KUKA KRL program: MyProgram_073().src

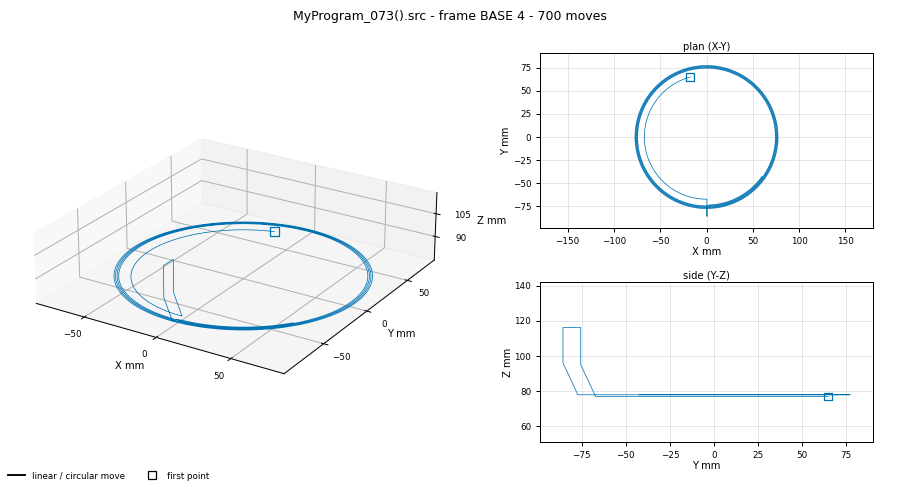
[picture p0: tool path of MyProgram_073().src in frame BASE 4, 700 of 700 moves have a stored position in this frame; points joined in program order, loops and branches not executed]
&ACCESS RVP
&REL 1
&PARAM TEMPLATE = C:\KRC\Roboter\Template\vorgabe
&PARAM EDITMASK = *
DEF MyProgram_073()
; ---- Setting reference (Base) ----
$BASE = BASE_DATA[4]

; --------------------------
; ---- Setting tool (TCP) ----
$TOOL = TOOL_DATA[3]
; --------------------------

$VEL.CP = VEL_APROX_PRINT
Startdeposition()
$VEL.CP = VEL_PRINT
LIN {X -17.4414,Y 64.8881,Z 77,A 99.3503,B 24.8705,C -2.6257,E1 24.9572,E2 344.7381} C_DIS
LIN {X -19.5195,Y 64.2946,Z 77,A 101.354,B 24.8704,C -2.6273,E1 24.9518,E2 342.7273} C_DIS
LIN {X -22.6182,Y 63.2711,Z 77,A 104.1504,B 24.8707,C -2.6243,E1 24.9445,E2 339.9329} C_DIS
LIN {X -25.654,Y 62.1019,Z 77,A 106.8913,B 24.8711,C -2.6198,E1 24.9374,E2 337.1966} C_DIS
LIN {X -27.9665,Y 61.0957,Z 77,A 109.0852,B 24.8714,C -2.6176,E1 24.9318,E2 335.0027} C_DIS
LIN {X -30.3307,Y 59.9565,Z 77,A 111.2597,B 24.8718,C -2.6126,E1 24.9263,E2 332.8342} C_DIS
LIN {X -32.9877,Y 58.5366,Z 77,A 113.6029,B 24.8728,C -2.6034,E1 24.9206,E2 330.5064} C_DIS
LIN {X -35.1348,Y 57.2737,Z 77,A 115.7355,B 24.8731,C -2.5997,E1 24.9155,E2 328.3759} C_DIS
LIN {X -37.2111,Y 55.947,Z 77,A 117.8448,B 24.8735,C -2.596,E1 24.9106,E2 326.2688} C_DIS
LIN {X -38.795,Y 54.8606,Z 77,A 119.7284,B 24.8733,C -2.598,E1 24.9063,E2 324.3738} C_DIS
LIN {X -41.2648,Y 53.028,Z 77,A 122.3339,B 24.8738,C -2.5922,E1 24.9005,E2 321.7728} C_DIS
LIN {X -43.4924,Y 51.216,Z 77,A 124.7333,B 24.8745,C -2.5859,E1 24.8953,E2 319.3795} C_DIS
LIN {X -45.7228,Y 49.2366,Z 77,A 127.4573,B 24.8747,C -2.5839,E1 24.8897,E2 316.6491} C_DIS
LIN {X -48.0153,Y 47.0029,Z 77,A 130.0891,B 24.8755,C -2.5754,E1 24.8845,E2 314.0265} C_DIS
LIN {X -50.0114,Y 44.8723,Z 77,A 132.6532,B 24.8759,C -2.5708,E1 24.8797,E2 311.462} C_DIS
LIN {X -51.9391,Y 42.6281,Z 77,A 135.2435,B 24.8764,C -2.5658,E1 24.875,E2 308.8718} C_DIS
LIN {X -53.955,Y 40.0458,Z 77,A 138.0531,B 24.8771,C -2.5588,E1 24.8703,E2 306.0656} C_DIS
LIN {X -55.8378,Y 37.3755,Z 77,A 140.854,B 24.8778,C -2.5515,E1 24.8659,E2 303.2682} C_DIS
LIN {X -57.2778,Y 35.128,Z 77,A 143.0663,B 24.8785,C -2.5438,E1 24.8626,E2 301.063} C_DIS
LIN {X -58.5282,Y 33.0027,Z 77,A 145.1855,B 24.8791,C -2.5382,E1 24.8597,E2 298.9463} C_DIS
LIN {X -59.947,Y 30.3494,Z 77,A 147.5323,B 24.8802,C -2.5262,E1 24.8566,E2 296.6154} C_DIS
LIN {X -61.0193,Y 28.1312,Z 77,A 149.6529,B 24.8808,C -2.5204,E1 24.8541,E2 294.4971} C_DIS
LIN {X -61.8116,Y 26.3449,Z 77,A 151.5592,B 24.8808,C -2.5204,E1 24.852,E2 292.5804} C_DIS
LIN {X -62.8919,Y 23.6492,Z 77,A 153.9533,B 24.8816,C -2.5112,E1 24.8496,E2 290.1948} C_DIS
LIN {X -63.8037,Y 21.0691,Z 77,A 156.4499,B 24.882,C -2.5074,E1 24.8473,E2 287.6931} C_DIS
LIN {X -64.5709,Y 18.583,Z 77,A 158.637,B 24.8827,C -2.4999,E1 24.8456,E2 285.5113} C_DIS
LIN {X -65.3372,Y 15.6772,Z 77,A 161.2488,B 24.8833,C -2.4929,E1 24.8438,E2 282.9009} C_DIS
LIN {X -65.9008,Y 13.1111,Z 77,A 163.5551,B 24.8839,C -2.4872,E1 24.8425,E2 280.5947} C_DIS
LIN {X -66.4404,Y 10.0194,Z 77,A 166.0408,B 24.885,C -2.4749,E1 24.8414,E2 278.1237} C_DIS
LIN {X -66.7829,Y 7.4076,Z 77,A 168.5127,B 24.8853,C -2.4724,E1 24.8406,E2 275.6429} C_DIS
LIN {X -67.0644,Y 4.1441,Z 77,A 171.3257,B 24.8861,C -2.4639,E1 24.84,E2 272.8332} C_DIS
LIN {X -67.1864,Y 0.8793,Z 77,A 174.1109,B 24.8869,C -2.4551,E1 24.8398,E2 270.0523} C_DIS
LIN {X -67.1706,Y -1.7002,Z 77,A 176.322,B 24.8875,C -2.4484,E1 24.8398,E2 267.844} C_DIS
LIN {X -67.01,Y -4.9472,Z 77,A 178.9028,B 24.8887,C -2.4357,E1 24.8403,E2 265.2779} C_DIS
LIN {X -66.7829,Y -7.4069,Z 77,A -178.7682,B 24.8888,C -2.4337,E1 24.841,E2 262.9398} C_DIS
LIN {X -66.4656,Y -9.8566,Z 77,A -176.8004,B 24.8897,C -2.4243,E1 24.8417,E2 260.9827} C_DIS
LIN {X -66.0524,Y -12.3243,Z 77,A -174.473,B 24.8899,C -2.4218,E1 24.8429,E2 258.6476} C_DIS
LIN {X -65.4042,Y -15.3955,Z 77,A -171.9941,B 24.891,C -2.4095,E1 24.8444,E2 256.1833} C_DIS
LIN {X -64.7607,Y -17.9129,Z 77,A -169.5742,B 24.8913,C -2.4071,E1 24.8461,E2 253.7552} C_DIS
LIN {X -64.0539,Y -20.2957,Z 77,A -167.6468,B 24.8922,C -2.3968,E1 24.8477,E2 251.8412} C_DIS
LIN {X -63.2656,Y -22.6337,Z 77,A -165.321,B 24.8923,C -2.3953,E1 24.8498,E2 249.5058} C_DIS
LIN {X -62.3396,Y -25.07,Z 77,A -163.1316,B 24.893,C -2.3883,E1 24.8521,E2 247.321} C_DIS
LIN {X -61.1455,Y -27.8561,Z 77,A -160.6723,B 24.8939,C -2.3784,E1 24.8548,E2 244.8718} C_DIS
LIN {X -60.0186,Y -30.2091,Z 77,A -158.2271,B 24.8939,C -2.3769,E1 24.8579,E2 242.417} C_DIS
LIN {X -58.6544,Y -32.7767,Z 77,A -155.7358,B 24.8946,C -2.3705,E1 24.8612,E2 239.9277} C_DIS
LIN {X -57.2052,Y -35.2475,Z 77,A -153.2924,B 24.8951,C -2.3642,E1 24.8647,E2 237.4869} C_DIS
LIN {X -55.7951,Y -37.4385,Z 77,A -151.1058,B 24.8957,C -2.3578,E1 24.8681,E2 235.3045} C_DIS
LIN {X -54.384,Y -39.4603,Z 77,A -148.9837,B 24.8961,C -2.3531,E1 24.8715,E2 233.1833} C_DIS
LIN {X -52.5036,Y -41.9302,Z 77,A -146.3519,B 24.8967,C -2.3465,E1 24.876,E2 230.5548} C_DIS
LIN {X -51.184,Y -43.53,Z 77,A -144.6169,B 24.8971,C -2.3418,E1 24.8791,E2 228.8231} C_DIS
LIN {X -49.2273,Y -45.7329,Z 77,A -141.9644,B 24.8973,C -2.3393,E1 24.8841,E2 226.1648} C_DIS
LIN {X -47.2236,Y -47.7973,Z 77,A -139.6629,B 24.8981,C -2.3309,E1 24.8886,E2 223.8736} C_DIS
LIN {X -45.1372,Y -49.774,Z 77,A -137.1132,B 24.8983,C -2.3281,E1 24.8939,E2 221.32} C_DIS
LIN {X -42.9447,Y -51.676,Z 77,A -134.7116,B 24.8988,C -2.3219,E1 24.899,E2 218.9241} C_DIS
LIN {X -40.6905,Y -53.4706,Z 77,A -132.0959,B 24.8989,C -2.321,E1 24.9047,E2 216.3008} C_DIS
LIN {X -38.6866,Y -54.9378,Z 77,A -129.9758,B 24.8992,C -2.3175,E1 24.9096,E2 214.1817} C_DIS
LIN {X -36.6463,Y -56.3194,Z 77,A -127.8662,B 24.8995,C -2.3145,E1 24.9145,E2 212.0724} C_DIS
LIN {X -34.5571,Y -57.6248,Z 77,A -125.8772,B 24.9,C -2.3089,E1 24.9192,E2 210.0906} C_DIS
LIN {X -32.3987,Y -58.8655,Z 77,A -123.6283,B 24.9,C -2.3089,E1 24.9247,E2 207.8352} C_DIS
LIN {X -30.2145,Y -60.0159,Z 77,A -121.5171,B 24.9002,C -2.3064,E1 24.9299,E2 205.7242} C_DIS
LIN {X -27.8627,Y -61.1425,Z 77,A -119.3351,B 24.9005,C -2.3029,E1 24.9355,E2 203.5449} C_DIS
LIN {X -25.0759,Y -62.3372,Z 77,A -116.8865,B 24.901,C -2.2972,E1 24.9418,E2 201.1044} C_DIS
LIN {X -22.6444,Y -63.2618,Z 77,A -114.4748,B 24.9008,C -2.2997,E1 24.9481,E2 198.6819} C_DIS
LIN {X -20.312,Y -64.0487,Z 77,A -112.5912,B 24.9013,C -2.2931,E1 24.9531,E2 196.8105} C_DIS
LIN {X -17.9227,Y -64.758,Z 77,A -110.242,B 24.901,C -2.2969,E1 24.9594,E2 194.4485} C_DIS
LIN {X -15.3953,Y -65.4043,Z 77,A -108.0635,B 24.9012,C -2.2947,E1 24.9653,E2 192.2723} C_DIS
LIN {X -12.4424,Y -66.0296,Z 77,A -105.7199,B 24.9018,C -2.2882,E1 24.9717,E2 189.9414} C_DIS
LIN {X -9.9977,Y -66.4438,Z 77,A -103.6077,B 24.9018,C -2.2876,E1 24.9775,E2 187.8287} C_DIS
LIN {X -7.5502,Y -66.7662,Z 77,A -101.2755,B 24.9014,C -2.2926,E1 24.984,E2 185.4829} C_DIS
LIN {X -4.954,Y -67.0095,Z 77,A -99.2056,B 24.9017,C -2.2889,E1 24.9898,E2 183.421} C_DIS
LIN {X -2.4711,Y -67.147,Z 77,A -96.8737,B 24.9013,C -2.2941,E1 24.9963,E2 181.076} C_DIS
LIN {X 0.4221,Y -67.1891,Z 77,A -94.9568,B 24.9024,C -2.2814,E1 25.0016,E2 179.1893} C_DIS
Enddeposition()
LIN {X 0.4386,Y -69.3021,Z 81.5315,A -94.9475,B 24.9027,C -2.2775,E1 25.0016,E2 179.1893} C_DIS
LIN {X 0.4882,Y -75.6412,Z 95.1262,A -94.9245,B 24.9035,C -2.2678,E1 25.0016,E2 179.1893} C_DIS
LIN {X 0.4882,Y -75.6412,Z 116.1262,A -95.2835,B 24.8902,C -2.4189,E1 25.0016,E2 179.1893} C_DIS
LIN {X 0.5081,Y -85.7186,Z 116.1262,A -95.3115,B 24.9057,C -2.2421,E1 25.0003,E2 179.6373} C_DIS
LIN {X 0.5081,Y -85.7186,Z 96.1262,A -94.9701,B 24.9174,C -2.0983,E1 25.0003,E2 179.6373} C_DIS
LIN {X 0.5081,Y -79.3793,Z 82.5315,A -94.9916,B 24.9167,C -2.1074,E1 25.0003,E2 179.6373} C_DIS
LIN {X 0.5081,Y -77.2663,Z 78,A -95.0003,B 24.9164,C -2.111,E1 25.0003,E2 179.6373} C_DIS
Startdeposition()
$VEL.CP = VEL_PRINT
LIN {X 3.5724,Y -77.1871,Z 78,A -91.8935,B 24.9145,C -2.1352,E1 25.0091,E2 176.4739} C_DIS
LIN {X 6.411,Y -77.0033,Z 78,A -89.9101,B 24.9147,C -2.1326,E1 25.0146,E2 174.4976} C_DIS
LIN {X 8.7348,Y -76.7744,Z 78,A -88.2092,B 24.9147,C -2.1326,E1 25.0194,E2 172.7976} C_DIS
LIN {X 10.6163,Y -76.5369,Z 78,A -86.6281,B 24.9142,C -2.1386,E1 25.0238,E2 171.2038} C_DIS
LIN {X 13.2103,Y -76.1331,Z 78,A -84.738,B 24.9142,C -2.1384,E1 25.029,E2 169.316} C_DIS
LIN {X 15.7888,Y -75.6394,Z 78,A -82.8059,B 24.9142,C -2.1396,E1 25.0343,E2 167.3833} C_DIS
LIN {X 18.0671,Y -75.1278,Z 78,A -80.9865,B 24.9138,C -2.1438,E1 25.0392,E2 165.5566} C_DIS
LIN {X 20.8201,Y -74.4119,Z 78,A -78.9095,B 24.9137,C -2.1451,E1 25.0448,E2 163.4798} C_DIS
LIN {X 23.3362,Y -73.6626,Z 78,A -77.0207,B 24.9137,C -2.1457,E1 25.0499,E2 161.5932} C_DIS
LIN {X 25.9989,Y -72.7653,Z 78,A -75.0657,B 24.9137,C -2.1445,E1 25.055,E2 159.6447} C_DIS
LIN {X 27.8093,Y -72.093,Z 78,A -73.5154,B 24.9133,C -2.1499,E1 25.0591,E2 158.085} C_DIS
LIN {X 29.7724,Y -71.3037,Z 78,A -72.0267,B 24.9133,C -2.1499,E1 25.0629,E2 156.6} C_DIS
LIN {X 32.1778,Y -70.2521,Z 78,A -69.914,B 24.9127,C -2.1576,E1 25.0683,E2 154.4739} C_DIS
LIN {X 34.7418,Y -69.0201,Z 78,A -67.9092,B 24.9127,C -2.1579,E1 25.0733,E2 152.4738} C_DIS
LIN {X 37.0659,Y -67.7992,Z 78,A -66.0648,B 24.9127,C -2.1582,E1 25.0779,E2 150.6339} C_DIS
LIN {X 38.9088,Y -66.7598,Z 78,A -64.5303,B 24.9125,C -2.16,E1 25.0816,E2 149.0999} C_DIS
LIN {X 40.7215,Y -65.6686,Z 78,A -62.792,B 24.9118,C -2.168,E1 25.0858,E2 147.3481} C_DIS
LIN {X 43.1109,Y -64.1253,Z 78,A -60.6916,B 24.9115,C -2.1718,E1 25.0907,E2 145.2456} C_DIS
LIN {X 45.265,Y -62.6246,Z 78,A -58.8065,B 24.9114,C -2.1739,E1 25.095,E2 143.3622} C_DIS
LIN {X 47.3656,Y -61.05,Z 78,A -56.7925,B 24.9109,C -2.1801,E1 25.0994,E2 141.3409} C_DIS
LIN {X 49.7493,Y -59.125,Z 78,A -54.6079,B 24.9107,C -2.1824,E1 25.1041,E2 139.1592} C_DIS
LIN {X 51.7284,Y -57.4001,Z 78,A -52.6061,B 24.9102,C -2.1885,E1 25.1083,E2 137.1508} C_DIS
LIN {X 53.964,Y -55.305,Z 78,A -50.411,B 24.9099,C -2.1915,E1 25.1128,E2 134.9576} C_DIS
LIN {X 55.4573,Y -53.8061,Z 78,A -48.9275,B 24.9099,C -2.1928,E1 25.1157,E2 133.4776} C_DIS
LIN {X 57.2538,Y -51.8918,Z 78,A -47.0377,B 24.9096,C -2.1959,E1 25.1192,E2 131.5887} C_DIS
LIN {X 58.5101,Y -50.4711,Z 78,A -45.6394,B 24.9093,C -2.1992,E1 25.1218,E2 130.1889} C_DIS
LIN {X 59.8692,Y -48.8496,Z 78,A -44.0797,B 24.909,C -2.203,E1 25.1246,E2 128.6273} C_DIS
LIN {X 61.05,Y -47.3656,Z 78,A -42.5054,B 24.9082,C -2.2119,E1 25.1273,E2 127.0395} C_DIS
LIN {X 62.6246,Y -45.265,Z 78,A -40.495,B 24.9076,C -2.2191,E1 25.1307,E2 125.0218} C_DIS
LIN {X 64.369,Y -42.7462,Z 78,A -38.4884,B 24.9078,C -2.2172,E1 25.1338,E2 123.0295} C_DIS
LIN {X 65.6686,Y -40.7215,Z 78,A -36.5637,B 24.907,C -2.2266,E1 25.1367,E2 121.0924} C_DIS
LIN {X 66.8691,Y -38.7186,Z 78,A -34.9946,B 24.907,C -2.2265,E1 25.1389,E2 119.5316} C_DIS
LIN {X 67.7992,Y -37.0659,Z 78,A -33.4212,B 24.9062,C -2.2357,E1 25.141,E2 117.9446} C_DIS
LIN {X 69.1843,Y -34.4106,Z 78,A -31.2395,B 24.9058,C -2.241,E1 25.1438,E2 115.7619} C_DIS
LIN {X 70.2521,Y -32.1778,Z 78,A -29.5677,B 24.9058,C -2.2414,E1 25.1458,E2 114.0982} C_DIS
LIN {X 71.0206,Y -30.4441,Z 78,A -28.1708,B 24.9054,C -2.2454,E1 25.1473,E2 112.6997} C_DIS
LIN {X 71.8265,Y -28.4878,Z 78,A -26.6126,B 24.905,C -2.2498,E1 25.149,E2 111.1396} C_DIS
LIN {X 72.6786,Y -26.2378,Z 78,A -24.8119,B 24.9045,C -2.2558,E1 25.1507,E2 109.3348} C_DIS
LIN {X 73.4383,Y -24.0297,Z 78,A -23.1208,B 24.9042,C -2.2599,E1 25.1522,E2 107.6437} C_DIS
LIN {X 74.0325,Y -22.1305,Z 78,A -21.4792,B 24.9034,C -2.2696,E1 25.1536,E2 105.9883} C_DIS
LIN {X 74.7736,Y -19.4812,Z 78,A -19.4536,B 24.9029,C -2.2756,E1 25.155,E2 103.9604} C_DIS
LIN {X 75.3932,Y -16.9301,Z 78,A -17.5731,B 24.9025,C -2.2796,E1 25.1562,E2 102.0812} C_DIS
LIN {X 75.9238,Y -14.359,Z 78,A -15.7346,B 24.9023,C -2.2824,E1 25.1572,E2 100.2468} C_DIS
LIN {X 76.323,Y -12.0583,Z 78,A -13.8679,B 24.9014,C -2.2921,E1 25.1581,E2 98.3681} C_DIS
LIN {X 76.6896,Y -9.4588,Z 78,A -11.9876,B 24.9011,C -2.2962,E1 25.1587,E2 96.4893} C_DIS
LIN {X 76.9188,Y -7.3554,Z 78,A -10.3392,B 24.9004,C -2.3037,E1 25.1592,E2 94.8329} C_DIS
LIN {X 77.1468,Y -4.3496,Z 78,A -8.1686,B 24.9,C -2.3089,E1 25.1596,E2 92.6631} C_DIS
LIN {X 77.2649,Y -0.9482,Z 78,A -5.7244,B 24.8995,C -2.3144,E1 25.1598,E2 90.2204} C_DIS
LIN {X 77.2557,Y 1.4489,Z 78,A -3.9631,B 24.8991,C -2.3196,E1 25.1598,E2 88.4573} C_DIS
LIN {X 77.1655,Y 4.0105,Z 78,A -2.1749,B 24.8988,C -2.3221,E1 25.1595,E2 86.6738} C_DIS
LIN {X 77.0033,Y 6.411,Z 78,A -0.3747,B 24.8983,C -2.3282,E1 25.1591,E2 84.8698} C_DIS
LIN {X 76.7744,Y 8.7348,Z 78,A 1.3165,B 24.8979,C -2.3324,E1 25.1586,E2 83.1787} C_DIS
LIN {X 76.5369,Y 10.6163,Z 78,A 2.7127,B 24.8976,C -2.3365,E1 25.1581,E2 81.7811} C_DIS
LIN {X 76.1693,Y 12.994,Z 78,A 4.6361,B 24.8967,C -2.3464,E1 25.1573,E2 79.8457} C_DIS
LIN {X 75.6394,Y 15.7888,Z 78,A 6.6081,B 24.8965,C -2.3486,E1 25.1562,E2 77.8799} C_DIS
LIN {X 75.0434,Y 18.413,Z 78,A 8.7541,B 24.8955,C -2.3593,E1 25.1548,E2 75.7209} C_DIS
LIN {X 74.4119,Y 20.8201,Z 78,A 10.5707,B 24.8951,C -2.364,E1 25.1535,E2 73.9038} C_DIS
LIN {X 73.6626,Y 23.3362,Z 78,A 12.4518,B 24.8948,C -2.3678,E1 25.1519,E2 72.0245} C_DIS
LIN {X 72.8689,Y 25.7037,Z 78,A 14.3528,B 24.8942,C -2.3748,E1 25.1502,E2 70.1177} C_DIS
LIN {X 71.8089,Y 28.5327,Z 78,A 16.536,B 24.8938,C -2.3795,E1 25.148,E2 67.9355} C_DIS
LIN {X 70.9329,Y 30.6451,Z 78,A 18.1646,B 24.8935,C -2.3822,E1 25.1462,E2 66.3093} C_DIS
LIN {X 69.8519,Y 33.0375,Z 78,A 20.0137,B 24.8933,C -2.3847,E1 25.1441,E2 64.4644} C_DIS
LIN {X 69.0201,Y 34.7418,Z 78,A 21.5348,B 24.8926,C -2.3921,E1 25.1422,E2 62.9339} C_DIS
LIN {X 67.7992,Y 37.0659,Z 78,A 23.4982,B 24.8921,C -2.3979,E1 25.1396,E2 60.9672} C_DIS
LIN {X 66.3889,Y 39.5363,Z 78,A 25.5956,B 24.8916,C -2.4031,E1 25.1366,E2 58.8683} C_DIS
LIN {X 65.164,Y 41.5242,Z 78,A 27.3414,B 24.8912,C -2.408,E1 25.134,E2 57.1197} C_DIS
LIN {X 63.5914,Y 43.8946,Z 78,A 29.2628,B 24.8912,C -2.4076,E1 25.131,E2 55.2087} C_DIS
LIN {X 62.1567,Y 45.904,Z 78,A 31.099,B 24.8908,C -2.4123,E1 25.128,E2 53.3704} C_DIS
LIN {X 60.9161,Y 47.5394,Z 78,A 32.5976,B 24.8905,C -2.4152,E1 25.1255,E2 51.8719} C_DIS
LIN {X 59.5909,Y 49.1887,Z 78,A 34.1584,B 24.8902,C -2.4186,E1 25.1227,E2 50.3103} C_DIS
LIN {X 58.0306,Y 51.0201,Z 78,A 36.0854,B 24.8895,C -2.427,E1 25.1192,E2 48.3723} C_DIS
LIN {X 56.1134,Y 53.1215,Z 78,A 38.1845,B 24.8891,C -2.4313,E1 25.1152,E2 46.2722} C_DIS
LIN {X 54.0086,Y 55.261,Z 78,A 40.2505,B 24.8891,C -2.4313,E1 25.1111,E2 44.2151} C_DIS
LIN {X 52.5905,Y 56.6127,Z 78,A 41.6938,B 24.8888,C -2.4339,E1 25.1082,E2 42.7713} C_DIS
LIN {X 51.1853,Y 57.8863,Z 78,A 43.094,B 24.8886,C -2.4365,E1 25.1053,E2 41.3707} C_DIS
LIN {X 49.5806,Y 59.2652,Z 78,A 44.8414,B 24.8878,C -2.4447,E1 25.1015,E2 39.6104} C_DIS
LIN {X 47.5394,Y 60.9161,Z 78,A 46.5952,B 24.888,C -2.4426,E1 25.0977,E2 37.8683} C_DIS
LIN {X 46.0301,Y 62.0644,Z 78,A 48.1194,B 24.8875,C -2.4485,E1 25.0943,E2 36.3356} C_DIS
LIN {X 44.313,Y 63.3006,Z 78,A 49.7356,B 24.8871,C -2.4525,E1 25.0906,E2 34.7154} C_DIS
LIN {X 41.9531,Y 64.8887,Z 78,A 51.8709,B 24.8867,C -2.4566,E1 25.0856,E2 32.5775} C_DIS
LIN {X 39.5363,Y 66.3889,Z 78,A 53.9546,B 24.8865,C -2.459,E1 25.0806,E2 30.4946} C_DIS
LIN {X 37.0659,Y 67.7992,Z 78,A 56.0713,B 24.8862,C -2.4621,E1 25.0755,E2 28.3768} C_DIS
LIN {X 34.7418,Y 69.0201,Z 78,A 57.9311,B 24.8862,C -2.4621,E1 25.0708,E2 26.5222} C_DIS
LIN {X 32.3767,Y 70.1595,Z 78,A 59.7773,B 24.8862,C -2.4615,E1 25.0662,E2 24.6822} C_DIS
LIN {X 30.214,Y 71.1176,Z 78,A 61.7043,B 24.8856,C -2.4684,E1 25.0612,E2 22.7435} C_DIS
LIN {X 27.6042,Y 72.1707,Z 78,A 63.7884,B 24.8855,C -2.4703,E1 25.0558,E2 20.6594} C_DIS
LIN {X 25.137,Y 73.0678,Z 78,A 65.6828,B 24.8855,C -2.4705,E1 25.0508,E2 18.7684} C_DIS
LIN {X 22.4305,Y 73.9435,Z 78,A 67.6298,B 24.8857,C -2.4675,E1 25.0457,E2 16.832} C_DIS
LIN {X 20.4809,Y 74.5063,Z 78,A 69.1796,B 24.8855,C -2.4698,E1 25.0415,E2 15.2793} C_DIS
LIN {X 18.0671,Y 75.1278,Z 78,A 71.1302,B 24.8851,C -2.4738,E1 25.0362,E2 13.3222} C_DIS
LIN {X 15.7888,Y 75.6394,Z 78,A 72.8846,B 24.8851,C -2.4752,E1 25.0314,E2 11.5666} C_DIS
LIN {X 13.2103,Y 76.1331,Z 78,A 74.8861,B 24.8848,C -2.4775,E1 25.0259,E2 9.562} C_DIS
LIN {X 10.3991,Y 76.5678,Z 78,A 76.7607,B 24.8854,C -2.4715,E1 25.0208,E2 7.7033} C_DIS
LIN {X 8.2988,Y 76.8227,Z 78,A 78.4702,B 24.885,C -2.4757,E1 25.016,E2 5.9851} C_DIS
LIN {X 5.6844,Y 77.0614,Z 78,A 80.2757,B 24.8853,C -2.4719,E1 25.011,E2 4.1896} C_DIS
LIN {X 3.5724,Y 77.1871,Z 78,A 82.0378,B 24.8848,C -2.4772,E1 25.006,E2 2.4156} C_DIS
LIN {X 0.7289,Y 77.2663,Z 78,A 84.134,B 24.8848,C -2.4765,E1 25.0002,E2 0.3211} C_DIS
LIN {X -2.1156,Y 77.2407,Z 78,A 86.2424,B 24.8849,C -2.476,E1 24.9943,E2 -1.7861} C_DIS
LIN {X -4.9571,Y 77.1105,Z 78,A 88.3533,B 24.885,C -2.4752,E1 24.9884,E2 -3.8959} C_DIS
LIN {X -7.5739,Y 76.8986,Z 78,A 90.3728,B 24.885,C -2.4763,E1 24.9828,E2 -5.9188} C_DIS
LIN {X -10.6163,Y 76.5369,Z 78,A 92.5774,B 24.8852,C -2.4731,E1 24.9767,E2 -8.1174} C_DIS
LIN {X -13.2103,Y 76.1331,Z 78,A 94.5292,B 24.8853,C -2.4718,E1 24.9713,E2 -10.0681} C_DIS
LIN {X -16.0036,Y 75.5953,Z 78,A 96.4626,B 24.8859,C -2.4654,E1 24.9661,E2 -11.9884} C_DIS
LIN {X -18.0671,Y 75.1278,Z 78,A 98.2126,B 24.8856,C -2.4688,E1 24.9613,E2 -13.7489} C_DIS
LIN {X -20.8201,Y 74.4119,Z 78,A 100.3265,B 24.8858,C -2.4668,E1 24.9556,E2 -15.8612} C_DIS
LIN {X -23.3465,Y 73.6593,Z 78,A 102.2266,B 24.8861,C -2.4631,E1 24.9506,E2 -17.7559} C_DIS
LIN {X -25.3439,Y 72.9951,Z 78,A 103.6735,B 24.8866,C -2.4583,E1 24.9467,E2 -19.194} C_DIS
LIN {X -27.6042,Y 72.1707,Z 78,A 105.6159,B 24.8864,C -2.4601,E1 24.9416,E2 -21.1448} C_DIS
LIN {X -29.7724,Y 71.3037,Z 78,A 107.3776,B 24.8866,C -2.4585,E1 24.9371,E2 -22.9066} C_DIS
LIN {X -32.3767,Y 70.1595,Z 78,A 109.4937,B 24.8868,C -2.4556,E1 24.9317,E2 -25.0208} C_DIS
LIN {X -34.7418,Y 69.0201,Z 78,A 111.5353,B 24.8868,C -2.4549,E1 24.9266,E2 -27.0663} C_DIS
LIN {X -37.4502,Y 67.5876,Z 78,A 113.7281,B 24.8874,C -2.4491,E1 24.9212,E2 -29.2513} C_DIS
LIN {X -39.7251,Y 66.2773,Z 78,A 115.6291,B 24.8879,C -2.4444,E1 24.9167,E2 -31.1469} C_DIS
LIN {X -41.9531,Y 64.8887,Z 78,A 117.6129,B 24.8881,C -2.4418,E1 24.912,E2 -33.1307} C_DIS
LIN {X -44.313,Y 63.3006,Z 78,A 119.6067,B 24.8888,C -2.4347,E1 24.9074,E2 -35.1145} C_DIS
LIN {X -46.2055,Y 61.9327,Z 78,A 121.4956,B 24.8888,C -2.4352,E1 24.9032,E2 -37.0111} C_DIS
LIN {X -48.4538,Y 60.19,Z 78,A 123.4366,B 24.8895,C -2.4264,E1 24.8989,E2 -38.9385} C_DIS
LIN {X -49.9163,Y 58.9828,Z 78,A 125.017,B 24.8894,C -2.4277,E1 24.8955,E2 -40.5281} C_DIS
LIN {X -52.0535,Y 57.1055,Z 78,A 126.9699,B 24.8902,C -2.419,E1 24.8915,E2 -42.468} C_DIS
LIN {X -53.4392,Y 55.8109,Z 78,A 128.5619,B 24.8901,C -2.4204,E1 24.8882,E2 -44.0699} C_DIS
LIN {X -55.305,Y 53.964,Z 78,A 130.3407,B 24.8909,C -2.4116,E1 24.8848,E2 -45.8351} C_DIS
LIN {X -56.6127,Y 52.5905,Z 78,A 131.8794,B 24.8909,C -2.4114,E1 24.8818,E2 -47.3801} C_DIS
LIN {X -58.0306,Y 51.0201,Z 78,A 133.5106,B 24.8911,C -2.4091,E1 24.8788,E2 -49.0131} C_DIS
LIN {X -59.7311,Y 49.02,Z 78,A 135.4149,B 24.8916,C -2.403,E1 24.8754,E2 -50.9117} C_DIS
LIN {X -61.05,Y 47.3656,Z 78,A 136.8683,B 24.8923,C -2.396,E1 24.8729,E2 -52.3553} C_DIS
LIN {X -62.194,Y 45.8531,Z 78,A 138.4614,B 24.8922,C -2.3969,E1 24.8702,E2 -53.9582} C_DIS
LIN {X -63.7166,Y 43.7145,Z 78,A 140.3665,B 24.8928,C -2.3906,E1 24.8672,E2 -55.8575} C_DIS
LIN {X -65.164,Y 41.5242,Z 78,A 142.3541,B 24.8931,C -2.3862,E1 24.8642,E2 -57.8447} C_DIS
LIN {X -66.3889,Y 39.5363,Z 78,A 144.1214,B 24.8935,C -2.3822,E1 24.8616,E2 -59.6116} C_DIS
LIN {X -67.7992,Y 37.0659,Z 78,A 146.2444,B 24.894,C -2.3765,E1 24.8588,E2 -61.7321} C_DIS
LIN {X -69.0201,Y 34.7418,Z 78,A 148.1501,B 24.8946,C -2.3698,E1 24.8563,E2 -63.6319} C_DIS
LIN {X -70.1595,Y 32.3767,Z 78,A 150.1386,B 24.895,C -2.3651,E1 24.854,E2 -65.62} C_DIS
LIN {X -71.3037,Y 29.7724,Z 78,A 152.299,B 24.8955,C -2.36,E1 24.8516,E2 -67.7803} C_DIS
LIN {X -72.4289,Y 26.9226,Z 78,A 154.396,B 24.8965,C -2.3488,E1 24.8495,E2 -69.8623} C_DIS
LIN {X -73.1378,Y 24.9291,Z 78,A 156.1507,B 24.8965,C -2.3486,E1 24.8479,E2 -71.6264} C_DIS
LIN {X -73.9435,Y 22.4305,Z 78,A 157.9361,B 24.8974,C -2.3386,E1 24.8464,E2 -73.3983} C_DIS
LIN {X -74.4717,Y 20.6091,Z 78,A 159.477,B 24.8974,C -2.3375,E1 24.8452,E2 -74.9455} C_DIS
LIN {X -75.1278,Y 18.0671,Z 78,A 161.341,B 24.8982,C -2.3294,E1 24.844,E2 -76.8011} C_DIS
LIN {X -75.6394,Y 15.7888,Z 78,A 163.2346,B 24.8983,C -2.3279,E1 24.8429,E2 -78.7023} C_DIS
LIN {X -76.1831,Y 12.9115,Z 78,A 165.4259,B 24.8989,C -2.3216,E1 24.8418,E2 -80.8914} C_DIS
LIN {X -76.6037,Y 10.1221,Z 78,A 167.5434,B 24.8994,C -2.3156,E1 24.841,E2 -83.0071} C_DIS
LIN {X -76.9188,Y 7.3554,Z 78,A 169.5752,B 24.9,C -2.3082,E1 24.8404,E2 -85.0335} C_DIS
LIN {X -77.1253,Y 4.7383,Z 78,A 171.5147,B 24.9006,C -2.3018,E1 24.84,E2 -86.9694} C_DIS
LIN {X -77.2407,Y 2.1156,Z 78,A 173.3794,B 24.9013,C -2.2936,E1 24.8398,E2 -88.8258} C_DIS
LIN {X -77.2697,Y -0.1952,Z 78,A 175.1003,B 24.9018,C -2.2884,E1 24.8398,E2 -90.5445} C_DIS
LIN {X -77.2407,Y -2.1156,Z 78,A 176.6893,B 24.9018,C -2.2879,E1 24.8398,E2 -92.1419} C_DIS
LIN {X -77.1105,Y -4.9571,Z 78,A 178.8134,B 24.9023,C -2.2816,E1 24.8402,E2 -94.2637} C_DIS
LIN {X -76.8986,Y -7.5739,Z 78,A -179.2797,B 24.9029,C -2.2745,E1 24.8407,E2 -96.1651} C_DIS
LIN {X -76.6614,Y -9.6763,Z 78,A -177.7717,B 24.9035,C -2.2681,E1 24.8412,E2 -97.6669} C_DIS
LIN {X -76.2895,Y -12.2751,Z 78,A -175.8646,B 24.9041,C -2.2611,E1 24.842,E2 -99.5685} C_DIS
LIN {X -75.9238,Y -14.359,Z 78,A -174.1061,B 24.9041,C -2.2609,E1 24.8429,E2 -101.3371} C_DIS
LIN {X -75.3932,Y -16.9301,Z 78,A -172.1694,B 24.9046,C -2.2547,E1 24.844,E2 -103.2703} C_DIS
LIN {X -74.719,Y -19.6937,Z 78,A -170.076,B 24.9052,C -2.2479,E1 24.8455,E2 -105.3598} C_DIS
LIN {X -74.0059,Y -22.2202,Z 78,A -168.212,B 24.9059,C -2.2401,E1 24.8469,E2 -107.2159} C_DIS
LIN {X -73.3006,Y -24.4463,Z 78,A -166.4981,B 24.9063,C -2.2345,E1 24.8484,E2 -108.9263} C_DIS
LIN {X -72.6786,Y -26.2378,Z 78,A -164.9043,B 24.9063,C -2.2351,E1 24.8499,E2 -110.5304} C_DIS
LIN {X -71.6636,Y -28.8951,Z 78,A -162.9595,B 24.9071,C -2.2249,E1 24.8519,E2 -112.4619} C_DIS
LIN {X -70.9329,Y -30.6451,Z 78,A -161.5442,B 24.9075,C -2.2211,E1 24.8534,E2 -113.8761} C_DIS
LIN {X -70.1595,Y -32.3767,Z 78,A -159.9511,B 24.9074,C -2.2219,E1 24.8553,E2 -115.4795} C_DIS
LIN {X -69.0201,Y -34.7418,Z 78,A -158.0458,B 24.9079,C -2.2155,E1 24.8576,E2 -117.3799} C_DIS
LIN {X -67.7992,Y -37.0659,Z 78,A -156.0763,B 24.9083,C -2.2108,E1 24.8602,E2 -119.3486} C_DIS
LIN {X -66.3889,Y -39.5363,Z 78,A -153.9367,B 24.9087,C -2.206,E1 24.8632,E2 -121.4879} C_DIS
LIN {X -64.8887,Y -41.9531,Z 78,A -151.8151,B 24.9091,C -2.2009,E1 24.8664,E2 -123.6082} C_DIS
LIN {X -63.3006,Y -44.313,Z 78,A -149.61,B 24.9094,C -2.1981,E1 24.8699,E2 -125.8174} C_DIS
LIN {X -61.4949,Y -46.7883,Z 78,A -147.5112,B 24.9102,C -2.1882,E1 24.8734,E2 -127.9027} C_DIS
LIN {X -59.8692,Y -48.8496,Z 78,A -145.4529,B 24.9103,C -2.1865,E1 24.877,E2 -129.9665} C_DIS
LIN {X -58.3658,Y -50.6363,Z 78,A -143.6878,B 24.9106,C -2.1834,E1 24.8802,E2 -131.7324} C_DIS
LIN {X -56.6127,Y -52.5905,Z 78,A -141.9095,B 24.9113,C -2.1748,E1 24.8835,E2 -133.4981} C_DIS
LIN {X -55.305,Y -53.964,Z 78,A -140.3721,B 24.9113,C -2.1752,E1 24.8865,E2 -135.043} C_DIS
LIN {X -53.8061,Y -55.4573,Z 78,A -138.7623,B 24.9114,C -2.173,E1 24.8897,E2 -136.6544} C_DIS
LIN {X -51.7284,Y -57.4001,Z 78,A -136.6122,B 24.9117,C -2.1699,E1 24.8941,E2 -138.8057} C_DIS
LIN {X -49.7493,Y -59.125,Z 78,A -134.7222,B 24.9121,C -2.1647,E1 24.8981,E2 -140.6907} C_DIS
LIN {X -47.97,Y -60.5757,Z 78,A -132.9969,B 24.9123,C -2.1622,E1 24.9019,E2 -142.4165} C_DIS
LIN {X -45.8531,Y -62.194,Z 78,A -130.976,B 24.9125,C -2.16,E1 24.9064,E2 -144.4394} C_DIS
LIN {X -43.7145,Y -63.7166,Z 78,A -128.9245,B 24.9125,C -2.1596,E1 24.9111,E2 -146.4968} C_DIS
LIN {X -41.0539,Y -65.461,Z 78,A -126.6654,B 24.913,C -2.1534,E1 24.9164,E2 -148.7484} C_DIS
LIN {X -38.7186,Y -66.8691,Z 78,A -124.804,B 24.9136,C -2.1462,E1 24.9209,E2 -150.5984} C_DIS
LIN {X -37.0659,Y -67.7992,Z 78,A -123.2157,B 24.9134,C -2.1492,E1 24.9248,E2 -152.1983} C_DIS
LIN {X -34.7418,Y -69.0201,Z 78,A -121.1752,B 24.9134,C -2.1492,E1 24.9299,E2 -154.2445} C_DIS
LIN {X -32.1778,Y -70.2521,Z 78,A -119.2649,B 24.914,C -2.1415,E1 24.9347,E2 -156.1412} C_DIS
LIN {X -29.7724,Y -71.3037,Z 78,A -117.2224,B 24.914,C -2.1421,E1 24.9399,E2 -158.1898} C_DIS
LIN {X -27.6042,Y -72.1707,Z 78,A -115.4624,B 24.914,C -2.1412,E1 24.9445,E2 -159.9515} C_DIS
LIN {X -25.137,Y -73.0678,Z 78,A -113.4073,B 24.914,C -2.1425,E1 24.9499,E2 -162.0137} C_DIS
LIN {X -22.2202,Y -74.0059,Z 78,A -111.2364,B 24.9143,C -2.1381,E1 24.9557,E2 -164.178} C_DIS
LIN {X -19.4812,Y -74.7736,Z 78,A -109.1245,B 24.9143,C -2.1369,E1 24.9614,E2 -166.2903} C_DIS
LIN {X -16.9301,Y -75.3932,Z 78,A -107.2287,B 24.9145,C -2.1345,E1 24.9666,E2 -168.1829} C_DIS
LIN {X -14.359,Y -75.9238,Z 78,A -105.3756,B 24.9148,C -2.1312,E1 24.9716,E2 -170.0302} C_DIS
LIN {X -12.0583,Y -76.323,Z 78,A -103.4945,B 24.9145,C -2.1348,E1 24.9768,E2 -171.9217} C_DIS
LIN {X -9.4588,Y -76.6896,Z 78,A -101.6001,B 24.9147,C -2.133,E1 24.9821,E2 -173.8131} C_DIS
LIN {X -7.3554,Y -76.9188,Z 78,A -99.9675,B 24.9145,C -2.1347,E1 24.9866,E2 -175.4505} C_DIS
LIN {X -4.7383,Y -77.1253,Z 78,A -98.0842,B 24.9147,C -2.1329,E1 24.9919,E2 -177.3303} C_DIS
LIN {X -2.1156,Y -77.2407,Z 78,A -96.1094,B 24.9146,C -2.1339,E1 24.9974,E2 -179.308} C_DIS
LIN {X 0.5081,Y -77.2663,Z 78,A -95.0001,B 24.9164,C -2.1109,E1 25.0003,E2 -180.3627} C_DIS
Enddeposition()
LIN {X 0.5081,Y -77.2663,Z 78,A -95.0001,B 24.9164,C -2.1109,E1 25.0003,E2 -180.3627} C_DIS
Startdeposition()
$VEL.CP = VEL_PRINT
LIN {X -0.888,Y -76.3341,Z 78,A -96.3437,B 24.9158,C -2.1189,E1 24.9966,E2 -179.038} C_DIS
LIN {X -4.0752,Y -76.2294,Z 78,A -98.6139,B 24.9155,C -2.1221,E1 24.9903,E2 -176.7747} C_DIS
LIN {X -7.3193,Y -75.987,Z 78,A -101.1784,B 24.9158,C -2.1188,E1 24.9831,E2 -174.2014} C_DIS
LIN {X -9.9543,Y -75.6865,Z 78,A -102.9935,B 24.9154,C -2.1239,E1 24.9781,E2 -172.397} C_DIS
LIN {X -12.7872,Y -75.2598,Z 78,A -105.2457,B 24.9156,C -2.1217,E1 24.9719,E2 -170.1377} C_DIS
LIN {X -15.7992,Y -74.6864,Z 78,A -107.588,B 24.9156,C -2.1216,E1 24.9655,E2 -167.7923} C_DIS
LIN {X -18.8711,Y -73.969,Z 78,A -109.7814,B 24.9151,C -2.1274,E1 24.9596,E2 -165.6099} C_DIS
LIN {X -20.6399,Y -73.4951,Z 78,A -111.1934,B 24.9151,C -2.1274,E1 24.9558,E2 -164.1953} C_DIS
LIN {X -23.3141,Y -72.6911,Z 78,A -113.3785,B 24.9151,C -2.1265,E1 24.9499,E2 -162.0044} C_DIS
LIN {X -26.7219,Y -71.5092,Z 78,A -116.8091,B 24.9165,C -2.11,E1 24.9408,E2 -158.5278} C_DIS
LIN {X -29.999,Y -70.1977,Z 78,A -118.7785,B 24.9149,C -2.1303,E1 24.9358,E2 -156.602} C_DIS
LIN {X -32.5947,Y -69.031,Z 78,A -120.925,B 24.9147,C -2.1324,E1 24.9304,E2 -154.4553} C_DIS
LIN {X -35.279,Y -67.6979,Z 78,A -123.1636,B 24.9145,C -2.1355,E1 24.9248,E2 -152.218} C_DIS
LIN {X -37.9349,Y -66.2455,Z 78,A -125.3876,B 24.9141,C -2.1398,E1 24.9194,E2 -149.9978} C_DIS
LIN {X -40.845,Y -64.4935,Z 78,A -128.8019,B 24.9156,C -2.1217,E1 24.9112,E2 -146.5297} C_DIS
LIN {X -44.001,Y -62.3827,Z 78,A -130.6068,B 24.9131,C -2.1526,E1 24.9072,E2 -144.7923} C_DIS
LIN {X -45.8586,Y -61.0287,Z 78,A -132.4701,B 24.9131,C -2.1521,E1 24.903,E2 -142.9211} C_DIS
LIN {X -48.0985,Y -59.2794,Z 78,A -134.6015,B 24.9128,C -2.156,E1 24.8984,E2 -140.791} C_DIS
LIN {X -50.2828,Y -57.4383,Z 78,A -136.7591,B 24.9125,C -2.1597,E1 24.8938,E2 -138.6339} C_DIS
LIN {X -52.3538,Y -55.5571,Z 78,A -138.9251,B 24.9123,C -2.1622,E1 24.8893,E2 -136.4652} C_DIS
LIN {X -54.8051,Y -53.141,Z 78,A -141.227,B 24.9113,C -2.1746,E1 24.8848,E2 -134.1831} C_DIS
LIN {X -56.295,Y -51.5596,Z 78,A -143.2637,B 24.9118,C -2.1681,E1 24.8809,E2 -132.1219} C_DIS
LIN {X -58.3294,Y -49.2474,Z 78,A -145.6223,B 24.9115,C -2.1722,E1 24.8766,E2 -129.7623} C_DIS
LIN {X -60.2886,Y -46.8282,Z 78,A -147.9267,B 24.911,C -2.1784,E1 24.8726,E2 -127.462} C_DIS
LIN {X -62.2985,Y -44.1189,Z 78,A -150.8726,B 24.9113,C -2.1746,E1 24.8678,E2 -124.4926} C_DIS
LIN {X -64.5432,Y -40.7656,Z 78,A -153.5535,B 24.91,C -2.1907,E1 24.8637,E2 -121.8366} C_DIS
LIN {X -66.1851,Y -38.04,Z 78,A -156.0477,B 24.9097,C -2.1944,E1 24.8602,E2 -119.3384} C_DIS
LIN {X -67.9512,Y -34.7872,Z 78,A -158.6332,B 24.9087,C -2.2066,E1 24.8568,E2 -116.7681} C_DIS
LIN {X -69.4152,Y -31.7685,Z 78,A -161.2145,B 24.9082,C -2.212,E1 24.8537,E2 -114.1858} C_DIS
LIN {X -70.5822,Y -29.0821,Z 78,A -163.4548,B 24.9078,C -2.2173,E1 24.8513,E2 -111.9457} C_DIS
LIN {X -71.4564,Y -26.8613,Z 78,A -165.1867,B 24.9072,C -2.2239,E1 24.8496,E2 -110.2197} C_DIS
LIN {X -72.4603,Y -24.0244,Z 78,A -167.5654,B 24.9069,C -2.2276,E1 24.8474,E2 -107.8364} C_DIS
LIN {X -73.8242,Y -19.4342,Z 78,A -171.1971,B 24.9061,C -2.2375,E1 24.8447,E2 -104.2072} C_DIS
LIN {X -74.5832,Y -16.2744,Z 78,A -174.3835,B 24.9069,C -2.2274,E1 24.8427,E2 -100.978} C_DIS
LIN {X -75.2963,Y -12.569,Z 78,A -176.7017,B 24.9052,C -2.2482,E1 24.8416,E2 -98.6957} C_DIS
LIN {X -75.7659,Y -9.3414,Z 78,A -178.9812,B 24.9042,C -2.2597,E1 24.8408,E2 -96.4302} C_DIS
LIN {X -76.0865,Y -6.1937,Z 78,A 178.6719,B 24.9035,C -2.2679,E1 24.8402,E2 -94.0887} C_DIS
LIN {X -76.2934,Y -2.6293,Z 78,A 175.6748,B 24.9035,C -2.2689,E1 24.8398,E2 -91.0759} C_DIS
LIN {X -76.3319,Y 1.0426,Z 78,A 173.1952,B 24.9021,C -2.2841,E1 24.8398,E2 -88.6177} C_DIS
LIN {X -76.0976,Y 6.0548,Z 78,A 169.9469,B 24.9,C -2.3083,E1 24.8403,E2 -85.4078} C_DIS
LIN {X -75.9086,Y 8.0879,Z 78,A 167.4138,B 24.9016,C -2.2897,E1 24.841,E2 -82.8149} C_DIS
LIN {X -75.4116,Y 11.8593,Z 78,A 165.0706,B 24.8998,C -2.3107,E1 24.842,E2 -80.508} C_DIS
LIN {X -74.8694,Y 14.9087,Z 78,A 162.621,B 24.8994,C -2.3151,E1 24.8432,E2 -78.0543} C_DIS
LIN {X -74.2588,Y 17.7005,Z 78,A 160.0047,B 24.8998,C -2.3108,E1 24.8449,E2 -75.4124} C_DIS
LIN {X -73.2989,Y 21.3293,Z 78,A 157.6195,B 24.8982,C -2.3297,E1 24.8467,E2 -73.0585} C_DIS
LIN {X -72.1891,Y 24.8287,Z 78,A 155.1181,B 24.8969,C -2.3441,E1 24.8488,E2 -70.5773} C_DIS
LIN {X -70.9456,Y 28.1838,Z 78,A 152.2406,B 24.8966,C -2.3478,E1 24.8517,E2 -67.6923} C_DIS
LIN {X -69.9461,Y 30.5787,Z 78,A 150.2495,B 24.8961,C -2.3526,E1 24.8539,E2 -65.7017} C_DIS
LIN {X -68.7175,Y 33.2485,Z 78,A 147.8184,B 24.8961,C -2.3538,E1 24.8568,E2 -63.2603} C_DIS
LIN {X -67.2914,Y 36.0492,Z 78,A 145.5875,B 24.8952,C -2.3636,E1 24.8597,E2 -61.041} C_DIS
LIN {X -64.9357,Y 40.1371,Z 78,A 142.3658,B 24.8936,C -2.3813,E1 24.8642,E2 -57.8447} C_DIS
LIN {X -63.5565,Y 42.2869,Z 78,A 140.1478,B 24.8938,C -2.3794,E1 24.8676,E2 -55.6111} C_DIS
LIN {X -61.0506,Y 45.8294,Z 78,A 136.3211,B 24.8942,C -2.3746,E1 24.8739,E2 -51.7543} C_DIS
LIN {X -58.4186,Y 49.1425,Z 78,A 133.6017,B 24.8925,C -2.3937,E1 24.8787,E2 -49.0679} C_DIS
LIN {X -55.106,Y 52.8288,Z 78,A 129.8875,B 24.8916,C -2.403,E1 24.8857,E2 -45.3596} C_DIS
LIN {X -51.2315,Y 56.5952,Z 78,A 126.0382,B 24.8903,C -2.4175,E1 24.8934,E2 -41.5289} C_DIS
LIN {X -49.1724,Y 58.3933,Z 78,A 123.7503,B 24.8904,C -2.4162,E1 24.8983,E2 -39.2291} C_DIS
LIN {X -46.8333,Y 60.2847,Z 78,A 120.5313,B 24.8921,C -2.3977,E1 24.9055,E2 -35.9541} C_DIS
LIN {X -43.3341,Y 62.8469,Z 78,A 118.4618,B 24.8889,C -2.4331,E1 24.9101,E2 -33.9619} C_DIS
LIN {X -40.9141,Y 64.4477,Z 78,A 115.7678,B 24.8897,C -2.4245,E1 24.9165,E2 -31.2386} C_DIS
LIN {X -36.3977,Y 67.1023,Z 78,A 112.1669,B 24.8883,C -2.4396,E1 24.9251,E2 -27.663} C_DIS
LIN {X -33.0541,Y 68.8109,Z 78,A 109.7064,B 24.8871,C -2.4531,E1 24.9312,E2 -25.2281} C_DIS
LIN {X -31.32,Y 69.6173,Z 78,A 107.8034,B 24.888,C -2.4434,E1 24.9361,E2 -23.2974} C_DIS
LIN {X -28.3611,Y 70.8757,Z 78,A 105.44,B 24.8875,C -2.448,E1 24.9422,E2 -20.9397} C_DIS
LIN {X -25.7393,Y 71.8693,Z 78,A 103.1868,B 24.8876,C -2.4469,E1 24.9481,E2 -18.6793} C_DIS
LIN {X -23.0571,Y 72.7743,Z 78,A 101.1725,B 24.8871,C -2.4522,E1 24.9534,E2 -16.6739} C_DIS
LIN {X -18.8448,Y 73.9757,Z 78,A 97.5661,B 24.8876,C -2.4474,E1 24.9632,E2 -13.0506} C_DIS
LIN {X -14.7134,Y 74.9073,Z 78,A 94.7401,B 24.8865,C -2.4592,E1 24.9708,E2 -10.2491} C_DIS
LIN {X -11.9005,Y 75.4052,Z 78,A 92.6403,B 24.8862,C -2.4619,E1 24.9766,E2 -8.1538} C_DIS
LIN {X -8.9968,Y 75.8062,Z 78,A 90.3676,B 24.8862,C -2.4613,E1 24.9829,E2 -5.878} C_DIS
LIN {X -5.5752,Y 76.1355,Z 78,A 87.7068,B 24.8864,C -2.4604,E1 24.9903,E2 -3.2138} C_DIS
LIN {X -2.4873,Y 76.2977,Z 78,A 85.5623,B 24.8859,C -2.4658,E1 24.9963,E2 -1.0817} C_DIS
LIN {X 0.1409,Y 76.3387,Z 78,A 83.464,B 24.8861,C -2.4629,E1 25.0022,E2 1.0235} C_DIS
LIN {X 3.1625,Y 76.2727,Z 78,A 81.3047,B 24.8859,C -2.466,E1 25.0082,E2 3.1748} C_DIS
LIN {X 5.8516,Y 76.1139,Z 78,A 79.0835,B 24.8864,C -2.4607,E1 25.0144,E2 5.4079} C_DIS
LIN {X 9.3135,Y 75.7691,Z 78,A 76.4612,B 24.8864,C -2.4599,E1 25.0217,E2 8.03} C_DIS
LIN {X 12.6397,Y 75.2845,Z 78,A 74.0832,B 24.8861,C -2.4631,E1 25.0282,E2 10.3982} C_DIS
LIN {X 15.8091,Y 74.6843,Z 78,A 71.516,B 24.8866,C -2.4581,E1 25.0352,E2 12.9742} C_DIS
LIN {X 18.9901,Y 73.9384,Z 78,A 69.2191,B 24.8863,C -2.461,E1 25.0414,E2 15.261} C_DIS
LIN {X 21.8157,Y 73.1546,Z 78,A 66.7815,B 24.8871,C -2.4529,E1 25.048,E2 17.7134} C_DIS
LIN {X 27.1508,Y 71.3468,Z 78,A 62.719,B 24.887,C -2.4538,E1 25.0587,E2 21.7656} C_DIS
LIN {X 30.1417,Y 70.1366,Z 78,A 60.369,B 24.887,C -2.4533,E1 25.0647,E2 24.1114} C_DIS
LIN {X 32.8179,Y 68.9244,Z 78,A 58.1611,B 24.8873,C -2.4507,E1 25.0703,E2 26.3199} C_DIS
LIN {X 35.5901,Y 67.5341,Z 78,A 55.9391,B 24.8873,C -2.4507,E1 25.0758,E2 28.5358} C_DIS
LIN {X 38.304,Y 66.0334,Z 78,A 53.4551,B 24.888,C -2.443,E1 25.0819,E2 31.0305} C_DIS
LIN {X 41.4786,Y 64.0868,Z 78,A 50.9267,B 24.8877,C -2.4463,E1 25.0879,E2 33.5429} C_DIS
LIN {X 43.9684,Y 62.4059,Z 78,A 48.4093,B 24.8887,C -2.4352,E1 25.0937,E2 36.0783} C_DIS
LIN {X 46.5631,Y 60.4929,Z 78,A 46.1662,B 24.8887,C -2.436,E1 25.0987,E2 38.3113} C_DIS
LIN {X 48.605,Y 58.8653,Z 78,A 44.1305,B 24.8892,C -2.4302,E1 25.1031,E2 40.353} C_DIS
LIN {X 50.8756,Y 56.9138,Z 78,A 41.9525,B 24.8894,C -2.4278,E1 25.1077,E2 42.528} C_DIS
LIN {X 53.2996,Y 54.6522,Z 78,A 39.6235,B 24.8894,C -2.4273,E1 25.1124,E2 44.8486} C_DIS
LIN {X 54.8963,Y 53.0464,Z 78,A 37.6345,B 24.8905,C -2.4153,E1 25.1163,E2 46.8574} C_DIS
LIN {X 56.9636,Y 50.82,Z 78,A 35.4355,B 24.8908,C -2.4127,E1 25.1204,E2 49.0531} C_DIS
LIN {X 58.7913,Y 48.6941,Z 78,A 33.3455,B 24.8912,C -2.4082,E1 25.1242,E2 51.1441} C_DIS
LIN {X 60.7518,Y 46.2271,Z 78,A 30.8777,B 24.8919,C -2.3996,E1 25.1284,E2 53.6207} C_DIS
LIN {X 62.9233,Y 43.2244,Z 78,A 28.4487,B 24.8916,C -2.403,E1 25.1323,E2 56.0296} C_DIS
LIN {X 64.352,Y 41.0655,Z 78,A 26.3256,B 24.8926,C -2.3928,E1 25.1356,E2 58.1663} C_DIS
LIN {X 66.0135,Y 38.3386,Z 78,A 23.8228,B 24.8934,C -2.3833,E1 25.1392,E2 60.6786} C_DIS
LIN {X 67.7363,Y 35.2062,Z 78,A 21.2021,B 24.8939,C -2.3779,E1 25.1426,E2 63.2983} C_DIS
LIN {X 69.0523,Y 32.5489,Z 78,A 19.0065,B 24.8944,C -2.3727,E1 25.1453,E2 65.4946} C_DIS
LIN {X 70.3153,Y 29.7199,Z 78,A 16.7893,B 24.8947,C -2.3693,E1 25.1478,E2 67.7076} C_DIS
LIN {X 71.5555,Y 26.5995,Z 78,A 14.436,B 24.8949,C -2.367,E1 25.1501,E2 70.0532} C_DIS
LIN {X 73.0225,Y 22.2567,Z 78,A 10.8705,B 24.8961,C -2.3531,E1 25.1533,E2 73.6315} C_DIS
LIN {X 73.7257,Y 19.8001,Z 78,A 9.0585,B 24.8963,C -2.3505,E1 25.1546,E2 75.4392} C_DIS
LIN {X 74.4261,Y 16.9796,Z 78,A 6.7471,B 24.8973,C -2.34,E1 25.1561,E2 77.7621} C_DIS
LIN {X 74.9947,Y 14.2598,Z 78,A 4.5981,B 24.898,C -2.3316,E1 25.1573,E2 79.9182} C_DIS
LIN {X 75.5061,Y 11.2481,Z 78,A 2.3456,B 24.8985,C -2.3257,E1 25.1583,E2 82.1715} C_DIS
LIN {X 75.9151,Y 8.0257,Z 78,A -0.0077,B 24.899,C -2.3206,E1 25.159,E2 84.5228} C_DIS
LIN {X 76.1738,Y 5.0088,Z 78,A -2.0885,B 24.899,C -2.3193,E1 25.1595,E2 86.5945} C_DIS
LIN {X 76.3182,Y 1.7837,Z 78,A -4.7135,B 24.9003,C -2.3055,E1 25.1598,E2 89.2366} C_DIS
LIN {X 76.3305,Y -1.1157,Z 78,A -6.878,B 24.9008,C -2.2989,E1 25.1598,E2 91.4036} C_DIS
LIN {X 76.2181,Y -4.2796,Z 78,A -9.115,B 24.9011,C -2.2956,E1 25.1595,E2 93.6352} C_DIS
LIN {X 75.989,Y -7.2986,Z 78,A -11.5092,B 24.9021,C -2.2846,E1 25.1589,E2 96.041} C_DIS
LIN {X 75.5999,Y -10.5915,Z 78,A -13.8761,B 24.9024,C -2.2804,E1 25.1581,E2 98.404} C_DIS
LIN {X 75.1386,Y -13.4798,Z 78,A -16.1099,B 24.9031,C -2.2723,E1 25.157,E2 100.6439} C_DIS
LIN {X 74.5235,Y -16.5483,Z 78,A -18.2665,B 24.9033,C -2.2707,E1 25.1558,E2 102.7917} C_DIS
LIN {X 73.8497,Y -19.3352,Z 78,A -20.5288,B 24.9041,C -2.2606,E1 25.1543,E2 105.0648} C_DIS
LIN {X 73.0864,Y -22.0456,Z 78,A -22.7757,B 24.905,C -2.2499,E1 25.1525,E2 107.3239} C_DIS
LIN {X 71.5237,Y -26.6834,Z 78,A -26.8757,B 24.9071,C -2.2258,E1 25.1486,E2 111.4579} C_DIS
LIN {X 69.4102,Y -31.7796,Z 78,A -30.5385,B 24.9069,C -2.2277,E1 25.1446,E2 115.0961} C_DIS
LIN {X 68.3572,Y -33.9824,Z 78,A -32.661,B 24.9081,C -2.2137,E1 25.1419,E2 117.2405} C_DIS
LIN {X 66.8964,Y -36.7772,Z 78,A -34.7391,B 24.9079,C -2.2154,E1 25.1392,E2 119.3036} C_DIS
LIN {X 65.3786,Y -39.411,Z 78,A -36.9148,B 24.9082,C -2.2121,E1 25.1361,E2 121.4759} C_DIS
LIN {X 63.6816,Y -42.0971,Z 78,A -39.3022,B 24.9088,C -2.2053,E1 25.1325,E2 123.8673} C_DIS
LIN {X 62.0486,Y -44.4692,Z 78,A -41.4458,B 24.9092,C -2.2,E1 25.129,E2 126.0131} C_DIS
LIN {X 59.6789,Y -47.6026,Z 78,A -44.301,B 24.9096,C -2.1949,E1 25.1242,E2 128.8668} C_DIS
LIN {X 57.7693,Y -49.9038,Z 78,A -46.5388,B 24.9101,C -2.1893,E1 25.1201,E2 131.1076} C_DIS
LIN {X 55.9879,Y -51.8942,Z 78,A -48.6134,B 24.9107,C -2.1822,E1 25.1162,E2 133.1898} C_DIS
LIN {X 53.7384,Y -54.2191,Z 78,A -50.909,B 24.9108,C -2.1803,E1 25.1117,E2 135.4802} C_DIS
LIN {X 51.888,Y -55.9936,Z 78,A -52.7961,B 24.9111,C -2.1769,E1 25.1079,E2 137.3676} C_DIS
LIN {X 49.9588,Y -57.7212,Z 78,A -54.8376,B 24.9117,C -2.1696,E1 25.1036,E2 139.4183} C_DIS
LIN {X 47.5801,Y -59.6971,Z 78,A -57.0959,B 24.912,C -2.1663,E1 25.0987,E2 141.6757} C_DIS
LIN {X 45.3373,Y -61.4177,Z 78,A -59.2285,B 24.9124,C -2.1616,E1 25.0939,E2 143.8118} C_DIS
LIN {X 42.4271,Y -63.4638,Z 78,A -62.0345,B 24.9131,C -2.1523,E1 25.0875,E2 146.6303} C_DIS
LIN {X 39.3396,Y -65.422,Z 78,A -64.7715,B 24.9135,C -2.1474,E1 25.0809,E2 149.3702} C_DIS
LIN {X 36.5551,Y -67.0169,Z 78,A -66.9476,B 24.9133,C -2.1499,E1 25.0757,E2 151.534} C_DIS
LIN {X 33.1879,Y -68.7466,Z 78,A -69.4412,B 24.9129,C -2.1553,E1 25.0695,E2 154.008} C_DIS
LIN {X 30.964,Y -69.7777,Z 78,A -72.6636,B 24.9163,C -2.113,E1 25.0611,E2 157.3226} C_DIS
LIN {X 27.0921,Y -71.369,Z 78,A -74.8043,B 24.9143,C -2.137,E1 25.0557,E2 159.4016} C_DIS
LIN {X 21.316,Y -73.3026,Z 78,A -79.429,B 24.9149,C -2.13,E1 25.0434,E2 164.0341} C_DIS
LIN {X 18.2632,Y -74.1215,Z 78,A -81.7887,B 24.9151,C -2.128,E1 25.037,E2 166.3951} C_DIS
LIN {X 15.3032,Y -74.7885,Z 78,A -84.3842,B 24.9159,C -2.1171,E1 25.0298,E2 169.0132} C_DIS
LIN {X 11.8026,Y -75.4204,Z 78,A -86.5971,B 24.9151,C -2.1278,E1 25.0238,E2 171.1984} C_DIS
LIN {X 9.0688,Y -75.7978,Z 78,A -88.8474,B 24.9156,C -2.1215,E1 25.0175,E2 173.4618} C_DIS
LIN {X 5.9273,Y -76.1078,Z 78,A -90.9835,B 24.9152,C -2.1267,E1 25.0116,E2 175.5842} C_DIS
LIN {X 3.1553,Y -76.273,Z 78,A -93.3203,B 24.9158,C -2.119,E1 25.0051,E2 177.9386} C_DIS
LIN {X 0.5091,Y -76.3356,Z 78,A -95.0941,B 24.9154,C -2.1243,E1 25.0001,E2 179.6997} C_DIS
Enddeposition()
LIN {X 0.5091,Y -76.3356,Z 78,A -95.0941,B 24.9154,C -2.1243,E1 25.0001,E2 179.6997} C_DIS
Startdeposition()
$VEL.CP = VEL_PRINT
LIN {X 2.9994,Y -75.3477,Z 78,A -92.553,B 24.9126,C -2.1588,E1 25.0075,E2 177.077} C_DIS
LIN {X 5.9692,Y -75.1704,Z 78,A -90.2203,B 24.9123,C -2.1618,E1 25.014,E2 174.7383} C_DIS
LIN {X 8.5048,Y -74.9263,Z 78,A -88.1242,B 24.9119,C -2.1673,E1 25.0198,E2 172.6304} C_DIS
LIN {X 11.4058,Y -74.5395,Z 78,A -85.6091,B 24.9111,C -2.177,E1 25.0268,E2 170.0946} C_DIS
LIN {X 15.9038,Y -73.711,Z 78,A -81.9038,B 24.9103,C -2.1865,E1 25.037,E2 166.3713} C_DIS
LIN {X 20.019,Y -72.7021,Z 78,A -78.9147,B 24.9106,C -2.1833,E1 25.0451,E2 163.3946} C_DIS
LIN {X 25.7332,Y -70.8804,Z 78,A -74.9312,B 24.9115,C -2.1724,E1 25.0556,E2 159.4444} C_DIS
LIN {X 30.2683,Y -69.0657,Z 78,A -71.2482,B 24.9111,C -2.1768,E1 25.0651,E2 155.7594} C_DIS
LIN {X 32.8044,Y -67.8978,Z 78,A -69.1506,B 24.9109,C -2.1794,E1 25.0704,E2 153.6611} C_DIS
LIN {X 36.187,Y -66.1573,Z 78,A -65.6586,B 24.9091,C -2.2017,E1 25.0791,E2 150.1261} C_DIS
LIN {X 39.5576,Y -64.1999,Z 78,A -62.8971,B 24.9091,C -2.2012,E1 25.0857,E2 147.3743} C_DIS
LIN {X 44.0897,Y -61.1754,Z 78,A -58.6357,B 24.9081,C -2.213,E1 25.0955,E2 143.0995} C_DIS
LIN {X 46.7942,Y -59.1314,Z 78,A -56.2942,B 24.9083,C -2.2116,E1 25.1007,E2 140.77} C_DIS
LIN {X 49.2813,Y -57.0767,Z 78,A -53.8138,B 24.9077,C -2.2179,E1 25.106,E2 138.2843} C_DIS
LIN {X 52.4178,Y -54.2089,Z 78,A -50.3452,B 24.9065,C -2.2326,E1 25.1131,E2 134.7951} C_DIS
LIN {X 54.5063,Y -52.1093,Z 78,A -48.3299,B 24.9066,C -2.231,E1 25.117,E2 132.7922} C_DIS
LIN {X 56.6976,Y -49.7154,Z 78,A -46.0263,B 24.9066,C -2.2324,E1 25.1213,E2 130.4956} C_DIS
LIN {X 59.4866,Y -46.3426,Z 78,A -42.3981,B 24.905,C -2.2502,E1 25.1277,E2 126.8423} C_DIS
LIN {X 62.1988,Y -42.6346,Z 78,A -39.3252,B 24.9053,C -2.2471,E1 25.1326,E2 123.7916} C_DIS
LIN {X 63.7067,Y -40.347,Z 78,A -37.0815,B 24.9044,C -2.2578,E1 25.136,E2 121.5339} C_DIS
LIN {X 65.805,Y -36.8229,Z 78,A -33.5024,B 24.9024,C -2.2807,E1 25.1411,E2 117.919} C_DIS
LIN {X 67.4952,Y -33.625,Z 78,A -31.0542,B 24.9025,C -2.2797,E1 25.1441,E2 115.4864} C_DIS
LIN {X 68.6082,Y -31.2929,Z 78,A -28.2701,B 24.8998,C -2.3106,E1 25.1474,E2 112.6443} C_DIS
LIN {X 70.3619,Y -27.1201,Z 78,A -26.1489,B 24.9024,C -2.2808,E1 25.1495,E2 110.6053} C_DIS
LIN {X 71.4857,Y -24.0003,Z 78,A -23.0711,B 24.9003,C -2.3055,E1 25.1523,E2 107.4864} C_DIS
LIN {X 72.4657,Y -20.8574,Z 78,A -20.0867,B 24.8983,C -2.3281,E1 25.1547,E2 104.4658} C_DIS
LIN {X 73.4444,Y -17.0923,Z 78,A -18.0285,B 24.8999,C -2.3099,E1 25.156,E2 102.4624} C_DIS
LIN {X 74.1407,Y -13.7678,Z 78,A -15.3628,B 24.899,C -2.3206,E1 25.1574,E2 99.787} C_DIS
LIN {X 74.6978,Y -10.3214,Z 78,A -12.8428,B 24.8986,C -2.325,E1 25.1585,E2 97.2714} C_DIS
LIN {X 75.0093,Y -7.7354,Z 78,A -10.6425,B 24.8974,C -2.3381,E1 25.1592,E2 95.0533} C_DIS
LIN {X 75.2571,Y -4.7639,Z 78,A -8.197,B 24.8963,C -2.3508,E1 25.1596,E2 92.5923} C_DIS
LIN {X 75.3926,Y -1.4777,Z 78,A -6.1213,B 24.8967,C -2.3458,E1 25.1598,E2 90.5408} C_DIS
LIN {X 75.3931,Y 1.4509,Z 78,A -3.8889,B 24.8961,C -2.3531,E1 25.1598,E2 88.3044} C_DIS
LIN {X 75.237,Y 5.0604,Z 78,A -1.0828,B 24.8952,C -2.3636,E1 25.1593,E2 85.4901} C_DIS
LIN {X 75.0078,Y 7.7491,Z 78,A 0.7975,B 24.8951,C -2.3649,E1 25.1588,E2 83.618} C_DIS
LIN {X 74.6289,Y 10.8066,Z 78,A 3.2402,B 24.8941,C -2.3753,E1 25.1579,E2 81.1651} C_DIS
LIN {X 74.024,Y 14.376,Z 78,A 6.1744,B 24.8929,C -2.3893,E1 25.1564,E2 78.2149} C_DIS
LIN {X 73.1003,Y 18.5104,Z 78,A 9.1309,B 24.8927,C -2.3912,E1 25.1545,E2 75.2712} C_DIS
LIN {X 72.3124,Y 21.3806,Z 78,A 11.9728,B 24.8905,C -2.4156,E1 25.1522,E2 72.3879} C_DIS
LIN {X 71.336,Y 24.4409,Z 78,A 13.5137,B 24.8923,C -2.3956,E1 25.1509,E2 70.9029} C_DIS
LIN {X 70.1651,Y 27.6238,Z 78,A 16.1388,B 24.8915,C -2.4045,E1 25.1484,E2 68.2715} C_DIS
LIN {X 69.1977,Y 29.9653,Z 78,A 18.2668,B 24.8905,C -2.416,E1 25.146,E2 66.1278} C_DIS
LIN {X 67.7267,Y 33.1577,Z 78,A 20.9831,B 24.8897,C -2.4248,E1 25.1428,E2 63.4054} C_DIS
LIN {X 66.3009,Y 35.9222,Z 78,A 24.0969,B 24.887,C -2.4537,E1 25.1386,E2 60.2395} C_DIS
LIN {X 64.3806,Y 39.2602,Z 78,A 26.6461,B 24.8873,C -2.45,E1 25.1349,E2 57.7121} C_DIS
LIN {X 62.3507,Y 42.4103,Z 78,A 29.8628,B 24.8857,C -2.4682,E1 25.1298,E2 54.4682} C_DIS
LIN {X 60.0432,Y 45.6201,Z 78,A 32.0892,B 24.8871,C -2.4524,E1 25.1262,E2 52.29} C_DIS
LIN {X 58.1243,Y 48.0398,Z 78,A 34.2706,B 24.8871,C -2.453,E1 25.1224,E2 50.1172} C_DIS
LIN {X 56.3446,Y 50.1154,Z 78,A 36.9759,B 24.8849,C -2.4762,E1 25.1173,E2 47.3693} C_DIS
LIN {X 53.9817,Y 52.6535,Z 78,A 39.1389,B 24.8857,C -2.4679,E1 25.1132,E2 45.2351} C_DIS
LIN {X 49.976,Y 56.4694,Z 78,A 43.0501,B 24.8857,C -2.4679,E1 25.1052,E2 41.3399} C_DIS
LIN {X 48.0479,Y 58.1175,Z 78,A 45.1844,B 24.8848,C -2.4775,E1 25.1006,E2 39.1911} C_DIS
LIN {X 45.5491,Y 60.0966,Z 78,A 47.9168,B 24.8836,C -2.4908,E1 25.0945,E2 36.4373} C_DIS
LIN {X 42.6592,Y 62.1821,Z 78,A 50.0263,B 24.8847,C -2.4781,E1 25.0898,E2 34.3652} C_DIS
LIN {X 40.9579,Y 63.3146,Z 78,A 52.575,B 24.8818,C -2.5091,E1 25.0836,E2 31.7513} C_DIS
LIN {X 37.7755,Y 65.2632,Z 78,A 54.8698,B 24.8829,C -2.4976,E1 25.0782,E2 29.4906} C_DIS
LIN {X 35.1684,Y 66.7038,Z 78,A 56.9157,B 24.8832,C -2.4945,E1 25.0732,E2 27.458} C_DIS
LIN {X 32.1797,Y 68.1971,Z 78,A 59.4286,B 24.883,C -2.4968,E1 25.0669,E2 24.9463} C_DIS
LIN {X 29.0006,Y 69.608,Z 78,A 61.845,B 24.8833,C -2.4933,E1 25.0607,E2 22.544} C_DIS
LIN {X 26.4923,Y 70.6005,Z 78,A 64.6552,B 24.8811,C -2.5165,E1 25.0533,E2 19.6848} C_DIS
LIN {X 21.6578,Y 72.2302,Z 78,A 67.8954,B 24.8825,C -2.5018,E1 25.0447,E2 16.4855} C_DIS
LIN {X 19.0958,Y 72.9498,Z 78,A 70.0524,B 24.882,C -2.5068,E1 25.0389,E2 14.32} C_DIS
LIN {X 14.8942,Y 73.9219,Z 78,A 73.3824,B 24.8818,C -2.5099,E1 25.0298,E2 10.9871} C_DIS
LIN {X 12.0022,Y 74.4467,Z 78,A 75.5075,B 24.882,C -2.5077,E1 25.024,E2 8.8695} C_DIS
LIN {X 8.9496,Y 74.8742,Z 78,A 77.7776,B 24.882,C -2.5063,E1 25.0177,E2 6.6047} C_DIS
LIN {X 5.0686,Y 75.2365,Z 78,A 81.124,B 24.8811,C -2.5168,E1 25.0083,E2 3.2349} C_DIS
LIN {X 1.6501,Y 75.3894,Z 78,A 83.3531,B 24.8821,C -2.5066,E1 25.0022,E2 1.0306} C_DIS
LIN {X -1.3442,Y 75.395,Z 78,A 85.7097,B 24.8819,C -2.5083,E1 24.9956,E2 -1.3301} C_DIS
LIN {X -6.0831,Y 75.1613,Z 78,A 89.1759,B 24.8824,C -2.5032,E1 24.986,E2 -4.7853} C_DIS
LIN {X -10.3443,Y 74.6946,Z 78,A 92.3317,B 24.8828,C -2.4987,E1 24.9772,E2 -7.9324} C_DIS
LIN {X -12.8331,Y 74.3081,Z 78,A 94.4897,B 24.8823,C -2.5037,E1 24.9712,E2 -10.1044} C_DIS
LIN {X -17.8663,Y 73.2599,Z 78,A 98.2976,B 24.8829,C -2.4977,E1 24.9609,E2 -13.9028} C_DIS
LIN {X -21.6159,Y 72.2426,Z 78,A 101.1586,B 24.8834,C -2.4923,E1 24.9532,E2 -16.7554} C_DIS
LIN {X -25.5594,Y 70.9432,Z 78,A 104.1801,B 24.8841,C -2.4851,E1 24.9453,E2 -19.7655} C_DIS
LIN {X -27.8244,Y 70.0863,Z 78,A 106.3835,B 24.8834,C -2.4919,E1 24.9395,E2 -21.9898} C_DIS
LIN {X -30.8905,Y 68.7896,Z 78,A 108.8921,B 24.8838,C -2.4877,E1 24.933,E2 -24.4942} C_DIS
LIN {X -35.98,Y 66.2696,Z 78,A 112.7576,B 24.8855,C -2.4695,E1 24.9235,E2 -28.3267} C_DIS
LIN {X -38.5646,Y 64.8,Z 78,A 115.6054,B 24.8845,C -2.4802,E1 24.9165,E2 -31.2085} C_DIS
LIN {X -41.8183,Y 62.7502,Z 78,A 118.2278,B 24.8858,C -2.4672,E1 24.9104,E2 -33.8084} C_DIS
LIN {X -43.5968,Y 61.5271,Z 78,A 120.0943,B 24.8855,C -2.4696,E1 24.9061,E2 -35.6869} C_DIS
LIN {X -46.2008,Y 59.5966,Z 78,A 122.727,B 24.8856,C -2.4687,E1 24.9003,E2 -38.327} C_DIS
LIN {X -49.6415,Y 56.7621,Z 78,A 125.9767,B 24.8866,C -2.4578,E1 24.8934,E2 -41.5633} C_DIS
LIN {X -52.6841,Y 53.9498,Z 78,A 129.2915,B 24.8869,C -2.4546,E1 24.8866,E2 -44.8841} C_DIS
LIN {X -55.5273,Y 51.019,Z 78,A 132.4758,B 24.8874,C -2.449,E1 24.8805,E2 -48.0689} C_DIS
LIN {X -57.7522,Y 48.4875,Z 78,A 134.7719,B 24.8886,C -2.436,E1 24.8764,E2 -50.3445} C_DIS
LIN {X -60.1846,Y 45.432,Z 78,A 138.1677,B 24.8884,C -2.4386,E1 24.8706,E2 -53.7627} C_DIS
LIN {X -62.4947,Y 42.1976,Z 78,A 141.1465,B 24.8892,C -2.4294,E1 24.8659,E2 -56.7341} C_DIS
LIN {X -64.2028,Y 39.5528,Z 78,A 143.5513,B 24.8898,C -2.423,E1 24.8623,E2 -59.1358} C_DIS
LIN {X -66.5725,Y 35.4177,Z 78,A 146.7406,B 24.8917,C -2.4022,E1 24.858,E2 -62.2923} C_DIS
LIN {X -68.3641,Y 31.8207,Z 78,A 149.857,B 24.8924,C -2.3947,E1 24.8542,E2 -65.4077} C_DIS
LIN {X -69.5863,Y 29.052,Z 78,A 152.1758,B 24.893,C -2.3883,E1 24.8517,E2 -67.7239} C_DIS
LIN {X -70.5905,Y 26.5186,Z 78,A 154.8416,B 24.8922,C -2.3962,E1 24.849,E2 -70.4236} C_DIS
LIN {X -71.9681,Y 22.5131,Z 78,A 157.4938,B 24.8944,C -2.3728,E1 24.8467,E2 -73.0351} C_DIS
LIN {X -72.826,Y 19.5603,Z 78,A 159.9028,B 24.8948,C -2.3673,E1 24.8449,E2 -75.4448} C_DIS
LIN {X -73.503,Y 16.8388,Z 78,A 162.8481,B 24.8937,C -2.38,E1 24.843,E2 -78.4379} C_DIS
LIN {X -74.2328,Y 13.2557,Z 78,A 164.6042,B 24.8967,C -2.3469,E1 24.8421,E2 -80.1253} C_DIS
LIN {X -74.7946,Y 9.5916,Z 78,A 168.2122,B 24.8958,C -2.3567,E1 24.8407,E2 -83.7783} C_DIS
LIN {X -75.2967,Y 4.078,Z 78,A 172.5532,B 24.8967,C -2.3465,E1 24.8399,E2 -88.1211} C_DIS
LIN {X -75.4033,Y 0.8421,Z 78,A 174.1421,B 24.8992,C -2.318,E1 24.8398,E2 -89.6513} C_DIS
LIN {X -75.3331,Y -3.3385,Z 78,A 177.3761,B 24.8999,C -2.3093,E1 24.84,E2 -92.8839} C_DIS
LIN {X -74.9569,Y -8.2356,Z 78,A -178.8373,B 24.9009,C -2.2988,E1 24.8409,E2 -96.6682} C_DIS
LIN {X -74.3659,Y -12.487,Z 78,A -175.4703,B 24.9015,C -2.2911,E1 24.8422,E2 -100.037} C_DIS
LIN {X -73.253,Y -17.8945,Z 78,A -171.2465,B 24.9026,C -2.2789,E1 24.8447,E2 -104.2566} C_DIS
LIN {X -71.9932,Y -22.4322,Z 78,A -167.8219,B 24.9038,C -2.2645,E1 24.8473,E2 -107.6666} C_DIS
LIN {X -71.3431,Y -24.4234,Z 78,A -165.8238,B 24.9034,C -2.2696,E1 24.8491,E2 -109.6881} C_DIS
LIN {X -70.1673,Y -27.6182,Z 78,A -162.7939,B 24.9031,C -2.2728,E1 24.8522,E2 -112.7429} C_DIS
LIN {X -68.4775,Y -31.5771,Z 78,A -159.9755,B 24.9048,C -2.2526,E1 24.8553,E2 -115.5286} C_DIS
LIN {X -66.9453,Y -34.7094,Z 78,A -156.6306,B 24.904,C -2.2624,E1 24.8596,E2 -118.9146} C_DIS
LIN {X -65.2937,Y -37.7223,Z 78,A -154.8767,B 24.9063,C -2.2345,E1 24.862,E2 -120.6111} C_DIS
LIN {X -63.8639,Y -40.0954,Z 78,A -152.4271,B 24.9061,C -2.2375,E1 24.8656,E2 -123.0803} C_DIS
LIN {X -61.3401,Y -43.859,Z 78,A -148.585,B 24.906,C -2.2388,E1 24.8717,E2 -126.9445} C_DIS
LIN {X -57.5338,Y -48.7455,Z 78,A -144.4191,B 24.908,C -2.2143,E1 24.879,E2 -131.0715} C_DIS
LIN {X -55.7026,Y -50.8279,Z 78,A -142.3303,B 24.9084,C -2.2092,E1 24.8828,E2 -133.1575} C_DIS
LIN {X -53.6399,Y -52.9997,Z 78,A -139.7917,B 24.9084,C -2.2109,E1 24.8878,E2 -135.7111} C_DIS
LIN {X -50.4845,Y -56.0142,Z 78,A -137.0251,B 24.91,C -2.1905,E1 24.8934,E2 -138.4403} C_DIS
LIN {X -48.8229,Y -57.4678,Z 78,A -134.3487,B 24.9082,C -2.2126,E1 24.8992,E2 -141.1797} C_DIS
LIN {X -46.2656,Y -59.5466,Z 78,A -132.6542,B 24.9102,C -2.1875,E1 24.9028,E2 -142.8207} C_DIS
LIN {X -44.4856,Y -60.8872,Z 78,A -130.8355,B 24.9102,C -2.1878,E1 24.9069,E2 -144.6466} C_DIS
LIN {X -40.6149,Y -63.5348,Z 78,A -127.2363,B 24.9106,C -2.1831,E1 24.9152,E2 -148.2465} C_DIS
LIN {X -38.1408,Y -65.0505,Z 78,A -124.9371,B 24.9106,C -2.1823,E1 24.9208,E2 -150.5509} C_DIS
LIN {X -35.3985,Y -66.5826,Z 78,A -122.5522,B 24.9109,C -2.1791,E1 24.9266,E2 -152.935} C_DIS
LIN {X -32.1518,Y -68.21,Z 78,A -119.7734,B 24.9112,C -2.1763,E1 24.9336,E2 -155.7144} C_DIS
LIN {X -29.3511,Y -69.4603,Z 78,A -116.9334,B 24.9103,C -2.1873,E1 24.941,E2 -158.587} C_DIS
LIN {X -24.727,Y -71.238,Z 78,A -113.7261,B 24.9117,C -2.1692,E1 24.9493,E2 -161.7579} C_DIS
LIN {X -21.9546,Y -72.1413,Z 78,A -111.4048,B 24.9117,C -2.1704,E1 24.9555,E2 -164.0861} C_DIS
LIN {X -18.0455,Y -73.2162,Z 78,A -108.3799,B 24.9119,C -2.1671,E1 24.9636,E2 -167.1077} C_DIS
LIN {X -15.1038,Y -73.8789,Z 78,A -106.0957,B 24.912,C -2.1659,E1 24.9699,E2 -169.3918} C_DIS
LIN {X -11.9307,Y -74.4583,Z 78,A -103.5952,B 24.912,C -2.1665,E1 24.9768,E2 -171.8961} C_DIS
LIN {X -8.3595,Y -74.9434,Z 78,A -100.7882,B 24.9118,C -2.1679,E1 24.9846,E2 -174.7084} C_DIS
LIN {X -5.1339,Y -75.232,Z 78,A -98.4466,B 24.9121,C -2.1646,E1 24.9911,E2 -177.0432} C_DIS
LIN {X -2.2888,Y -75.3723,Z 78,A -96.422,B 24.9124,C -2.161,E1 24.9967,E2 -179.0597} C_DIS
LIN {X 0.5052,Y -75.4053,Z 78,A -95.2376,B 24.9144,C -2.1359,E1 24.9998,E2 -180.1846} C_DIS
Enddeposition()
LIN {X 0.5052,Y -75.4053,Z 78,A -95.2376,B 24.9144,C -2.1359,E1 24.9998,E2 -180.1846} C_DIS
Startdeposition()
$VEL.CP = VEL_PRINT
LIN {X -0.1965,Y -74.4761,Z 78,A -95.8218,B 24.9132,C -2.1509,E1 24.9983,E2 -179.636} C_DIS
LIN {X -3.1805,Y -74.4079,Z 78,A -98.1456,B 24.9133,C -2.1499,E1 24.9918,E2 -177.3094} C_DIS
LIN {X -5.7163,Y -74.2565,Z 78,A -100.2579,B 24.9136,C -2.1458,E1 24.9859,E2 -175.1863} C_DIS
LIN {X -10.8054,Y -73.6886,Z 78,A -104.0809,B 24.9133,C -2.1495,E1 24.9753,E2 -171.3695} C_DIS
LIN {X -13.9914,Y -73.1499,Z 78,A -106.477,B 24.9131,C -2.1526,E1 24.9687,E2 -168.9785} C_DIS
LIN {X -17.2155,Y -72.4594,Z 78,A -109.809,B 24.9146,C -2.1335,E1 24.9595,E2 -165.5966} C_DIS
LIN {X -20.7448,Y -71.5298,Z 78,A -111.8585,B 24.9129,C -2.1546,E1 24.9542,E2 -163.594} C_DIS
LIN {X -24.5189,Y -70.3242,Z 78,A -115.0587,B 24.9131,C -2.1531,E1 24.9456,E2 -160.3844} C_DIS
LIN {X -28.7031,Y -68.7229,Z 78,A -118.4225,B 24.9126,C -2.1585,E1 24.9369,E2 -157.0261} C_DIS
LIN {X -31.709,Y -67.3891,Z 78,A -121.4334,B 24.9134,C -2.1493,E1 24.9292,E2 -153.9859} C_DIS
LIN {X -35.7864,Y -65.3153,Z 78,A -124.4847,B 24.912,C -2.1655,E1 24.9218,E2 -150.9645} C_DIS
LIN {X -37.8844,Y -64.1204,Z 78,A -126.8166,B 24.9128,C -2.1564,E1 24.9161,E2 -148.6039} C_DIS
LIN {X -42.668,Y -61.0421,Z 78,A -130.7398,B 24.9113,C -2.1744,E1 24.907,E2 -144.7106} C_DIS
LIN {X -44.477,Y -59.7373,Z 78,A -132.4012,B 24.911,C -2.1786,E1 24.9033,E2 -143.0535} C_DIS
LIN {X -48.0934,Y -56.8661,Z 78,A -135.9444,B 24.9104,C -2.1853,E1 24.8956,E2 -139.5129} C_DIS
LIN {X -50.9179,Y -54.3511,Z 78,A -139.1337,B 24.9105,C -2.1843,E1 24.889,E2 -136.3083} C_DIS
LIN {X -54.0743,Y -51.2122,Z 78,A -142.3471,B 24.9095,C -2.1966,E1 24.8828,E2 -133.1105} C_DIS
LIN {X -55.9196,Y -49.1907,Z 78,A -144.3831,B 24.909,C -2.2029,E1 24.879,E2 -131.0806} C_DIS
LIN {X -58.0375,Y -46.6731,Z 78,A -146.9984,B 24.9087,C -2.2068,E1 24.8743,E2 -128.4623} C_DIS
LIN {X -59.7556,Y -44.4527,Z 78,A -149.266,B 24.9084,C -2.2094,E1 24.8705,E2 -126.1901} C_DIS
LIN {X -61.7054,Y -41.7026,Z 78,A -152.0803,B 24.9084,C -2.2107,E1 24.866,E2 -123.3649} C_DIS
LIN {X -63.8411,Y -38.3551,Z 78,A -154.6397,B 24.9067,C -2.2302,E1 24.8623,E2 -120.8391} C_DIS
LIN {X -65.5183,Y -35.4122,Z 78,A -157.9663,B 24.9075,C -2.2203,E1 24.8577,E2 -117.4714} C_DIS
LIN {X -67.3543,Y -31.7837,Z 78,A -161.0461,B 24.9067,C -2.2301,E1 24.854,E2 -114.3982} C_DIS
LIN {X -69.1642,Y -27.6252,Z 78,A -164.519,B 24.9058,C -2.2404,E1 24.8503,E2 -110.9306} C_DIS
LIN {X -70.6026,Y -23.705,Z 78,A -167.2207,B 24.904,C -2.2616,E1 24.8478,E2 -108.2641} C_DIS
LIN {X -71.7658,Y -19.9084,Z 78,A -170.6457,B 24.904,C -2.2621,E1 24.8451,E2 -104.8208} C_DIS
LIN {X -72.4994,Y -17.0461,Z 78,A -172.9961,B 24.9036,C -2.2673,E1 24.8435,E2 -102.4688} C_DIS
LIN {X -73.2576,Y -13.4179,Z 78,A -175.7446,B 24.9026,C -2.2784,E1 24.8421,E2 -99.7306} C_DIS
LIN {X -73.9319,Y -8.9906,Z 78,A -178.7815,B 24.9009,C -2.2985,E1 24.8409,E2 -96.7235} C_DIS
LIN {X -74.2414,Y -5.905,Z 78,A 178.3759,B 24.9011,C -2.2955,E1 24.8401,E2 -93.8569} C_DIS
LIN {X -74.4423,Y -2.2361,Z 78,A 175.3498,B 24.9008,C -2.2999,E1 24.8398,E2 -90.823} C_DIS
LIN {X -74.4558,Y 1.7768,Z 78,A 171.6061,B 24.9012,C -2.2949,E1 24.84,E2 -87.0449} C_DIS
LIN {X -74.2446,Y 5.865,Z 78,A 169.6742,B 24.8979,C -2.3325,E1 24.8404,E2 -85.1911} C_DIS
LIN {X -73.8785,Y 9.4151,Z 78,A 166.2037,B 24.8986,C -2.3247,E1 24.8415,E2 -81.6813} C_DIS
LIN {X -73.2564,Y 13.4243,Z 78,A 162.827,B 24.8982,C -2.3288,E1 24.8431,E2 -78.2943} C_DIS
LIN {X -72.5916,Y 16.6472,Z 78,A 160.7595,B 24.8966,C -2.3472,E1 24.8443,E2 -76.2587} C_DIS
LIN {X -71.4307,Y 21.079,Z 78,A 157.5407,B 24.895,C -2.3652,E1 24.8467,E2 -73.064} C_DIS
LIN {X -70.5248,Y 23.9358,Z 78,A 154.8726,B 24.8951,C -2.364,E1 24.849,E2 -70.3779} C_DIS
LIN {X -68.8463,Y 28.4072,Z 78,A 151.3128,B 24.8939,C -2.3777,E1 24.8526,E2 -66.8309} C_DIS
LIN {X -67.5596,Y 31.3426,Z 78,A 148.1462,B 24.8947,C -2.3691,E1 24.8563,E2 -63.6265} C_DIS
LIN {X -65.9998,Y 34.507,Z 78,A 146.2231,B 24.8924,C -2.3951,E1 24.8587,E2 -61.755} C_DIS
LIN {X -63.4688,Y 38.9676,Z 78,A 142.4498,B 24.891,C -2.4103,E1 24.864,E2 -57.9984} C_DIS
LIN {X -61.1938,Y 42.4497,Z 78,A 139.24,B 24.8902,C -2.4189,E1 24.8689,E2 -54.793} C_DIS
LIN {X -58.9388,Y 45.5289,Z 78,A 135.4778,B 24.8912,C -2.4075,E1 24.8753,E2 -50.9857} C_DIS
LIN {X -55.5916,Y 49.5606,Z 78,A 131.9497,B 24.8892,C -2.4295,E1 24.8816,E2 -47.4938} C_DIS
LIN {X -53.4895,Y 51.8224,Z 78,A 129.5165,B 24.8888,C -2.4339,E1 24.8863,E2 -45.0606} C_DIS
LIN {X -51.1528,Y 54.1302,Z 78,A 126.8115,B 24.8887,C -2.4356,E1 24.8917,E2 -42.3485} C_DIS
LIN {X -47.8779,Y 57.0467,Z 78,A 123.1009,B 24.8887,C -2.4352,E1 24.8996,E2 -38.6224} C_DIS
LIN {X -44.7157,Y 59.5581,Z 78,A 120.6767,B 24.8866,C -2.4579,E1 24.9049,E2 -36.2436} C_DIS
LIN {X -42.4617,Y 61.1855,Z 78,A 118.3516,B 24.8866,C -2.4577,E1 24.9102,E2 -33.9099} C_DIS
LIN {X -39.2612,Y 63.2871,Z 78,A 114.9467,B 24.8871,C -2.4522,E1 24.9183,E2 -30.4811} C_DIS
LIN {X -36.0328,Y 65.1797,Z 78,A 112.1651,B 24.8865,C -2.4595,E1 24.925,E2 -27.7088} C_DIS
LIN {X -31.7514,Y 67.3693,Z 78,A 108.732,B 24.8853,C -2.4718,E1 24.9336,E2 -24.2959} C_DIS
LIN {X -28.7554,Y 68.7009,Z 78,A 106.0813,B 24.8853,C -2.4723,E1 24.9404,E2 -21.6402} C_DIS
LIN {X -22.8952,Y 70.8693,Z 78,A 101.9138,B 24.8832,C -2.4942,E1 24.9512,E2 -17.5164} C_DIS
LIN {X -20.688,Y 71.5459,Z 78,A 99.2651,B 24.8851,C -2.4744,E1 24.9584,E2 -14.8163} C_DIS
LIN {X -16.5993,Y 72.6027,Z 78,A 95.8917,B 24.8851,C -2.4744,E1 24.9676,E2 -11.4381} C_DIS
LIN {X -11.9292,Y 73.5151,Z 78,A 91.5986,B 24.8863,C -2.4613,E1 24.9795,E2 -7.1099} C_DIS
LIN {X -7.3101,Y 74.1176,Z 78,A 89.3687,B 24.8829,C -2.4973,E1 24.9855,E2 -4.9641} C_DIS
LIN {X -2.0139,Y 74.4491,Z 78,A 85.0178,B 24.8834,C -2.4919,E1 24.9976,E2 -0.5992} C_DIS
LIN {X 0.3222,Y 74.4753,Z 78,A 82.8907,B 24.8842,C -2.4838,E1 25.0036,E2 1.5471} C_DIS
LIN {X 4.2802,Y 74.353,Z 78,A 79.5036,B 24.885,C -2.4752,E1 25.0131,E2 4.9536} C_DIS
LIN {X 7.7353,Y 74.0731,Z 78,A 77.5159,B 24.8834,C -2.4924,E1 25.0185,E2 6.899} C_DIS
LIN {X 10.7425,Y 73.6975,Z 78,A 75.0937,B 24.8837,C -2.4895,E1 25.0252,E2 9.326} C_DIS
LIN {X 13.9722,Y 73.1536,Z 78,A 71.8488,B 24.8855,C -2.4696,E1 25.0343,E2 12.6146} C_DIS
LIN {X 17.746,Y 72.3308,Z 78,A 69.7401,B 24.8836,C -2.4907,E1 25.0399,E2 14.6702} C_DIS
LIN {X 21.416,Y 71.3305,Z 78,A 66.6581,B 24.8841,C -2.4845,E1 25.0482,E2 17.7617} C_DIS
LIN {X 25.8326,Y 69.853,Z 78,A 63.2534,B 24.884,C -2.4862,E1 25.0571,E2 21.1556} C_DIS
LIN {X 28.6147,Y 68.7602,Z 78,A 60.5094,B 24.8853,C -2.4719,E1 25.0643,E2 23.9271} C_DIS
LIN {X 32.6751,Y 66.9268,Z 78,A 57.4289,B 24.8848,C -2.4773,E1 25.072,E2 26.987} C_DIS
LIN {X 35.9289,Y 65.2369,Z 78,A 54.5793,B 24.8852,C -2.4728,E1 25.079,E2 29.8392} C_DIS
LIN {X 40.2784,Y 62.6443,Z 78,A 50.7973,B 24.8855,C -2.4701,E1 25.088,E2 33.6156} C_DIS
LIN {X 42.9189,Y 60.867,Z 78,A 47.6096,B 24.8877,C -2.4457,E1 25.0954,E2 36.8502} C_DIS
LIN {X 45.8545,Y 58.6872,Z 78,A 45.5197,B 24.8864,C -2.4607,E1 25.1,E2 38.897} C_DIS
LIN {X 47.6179,Y 57.2642,Z 78,A 43.0746,B 24.8885,C -2.4379,E1 25.1053,E2 41.3865} C_DIS
LIN {X 50.3653,Y 54.8634,Z 78,A 40.8065,B 24.8876,C -2.4473,E1 25.1099,E2 43.6232} C_DIS
LIN {X 53.351,Y 51.9662,Z 78,A 36.7447,B 24.8904,C -2.4165,E1 25.118,E2 47.7406} C_DIS
LIN {X 56.4639,Y 48.5655,Z 78,A 34.2965,B 24.8883,C -2.4394,E1 25.1224,E2 50.1237} C_DIS
LIN {X 58.1414,Y 46.545,Z 78,A 31.8421,B 24.8899,C -2.4223,E1 25.1267,E2 52.607} C_DIS
LIN {X 61.6677,Y 41.7581,Z 78,A 28.0475,B 24.8889,C -2.4334,E1 25.1328,E2 56.3571} C_DIS
LIN {X 63.0285,Y 39.6753,Z 78,A 26.2313,B 24.8891,C -2.4313,E1 25.1356,E2 58.1691} C_DIS
LIN {X 64.1647,Y 37.8095,Z 78,A 23.6686,B 24.8918,C -2.4015,E1 25.1393,E2 60.7891} C_DIS
LIN {X 66.2898,Y 33.9457,Z 78,A 20.7921,B 24.8913,C -2.4072,E1 25.143,E2 63.637} C_DIS
LIN {X 67.2803,Y 31.9395,Z 78,A 18.7689,B 24.8925,C -2.3936,E1 25.1455,E2 65.6814} C_DIS
LIN {X 68.9524,Y 28.1464,Z 78,A 16.0884,B 24.892,C -2.3993,E1 25.1484,E2 68.3336} C_DIS
LIN {X 70.1256,Y 25.085,Z 78,A 12.8832,B 24.8944,C -2.3721,E1 25.1515,E2 71.5852} C_DIS
LIN {X 71.6728,Y 20.2402,Z 78,A 9.5509,B 24.8939,C -2.3774,E1 25.1542,E2 74.8861} C_DIS
LIN {X 72.2934,Y 17.8993,Z 78,A 7.0036,B 24.8962,C -2.3518,E1 25.156,E2 77.4791} C_DIS
LIN {X 73.0534,Y 14.4922,Z 78,A 4.5323,B 24.8964,C -2.3497,E1 25.1573,E2 79.9408} C_DIS
LIN {X 73.7829,Y 10.1419,Z 78,A 1.6024,B 24.8961,C -2.3528,E1 25.1585,E2 82.8464} C_DIS
LIN {X 74.0687,Y 7.7773,Z 78,A -0.5708,B 24.8975,C -2.337,E1 25.1592,E2 85.0439} C_DIS
LIN {X 74.4452,Y 2.1421,Z 78,A -4.4457,B 24.8975,C -2.3371,E1 25.1598,E2 88.8956} C_DIS
LIN {X 74.4725,Y -0.7891,Z 78,A -6.4102,B 24.8974,C -2.3385,E1 25.1598,E2 90.8451} C_DIS
LIN {X 74.3098,Y -4.9715,Z 78,A -9.5009,B 24.898,C -2.3321,E1 25.1594,E2 93.9325} C_DIS
LIN {X 73.9574,Y -8.7731,Z 78,A -12.7855,B 24.8997,C -2.3124,E1 25.1585,E2 97.2441} C_DIS
LIN {X 73.5317,Y -11.8299,Z 78,A -15.2554,B 24.9006,C -2.3021,E1 25.1575,E2 99.724} C_DIS
LIN {X 73.0455,Y -14.5328,Z 78,A -17.5246,B 24.9015,C -2.2908,E1 25.1563,E2 102.0066} C_DIS
LIN {X 72.0991,Y -18.6652,Z 78,A -20.709,B 24.9022,C -2.2828,E1 25.1542,E2 105.1915} C_DIS
LIN {X 71.1502,Y -22.0068,Z 78,A -23.3239,B 24.9028,C -2.2762,E1 25.1521,E2 107.807} C_DIS
LIN {X 69.9384,Y -25.5985,Z 78,A -25.8557,B 24.9026,C -2.2786,E1 25.1498,E2 110.319} C_DIS
LIN {X 69.2802,Y -27.3297,Z 78,A -28.2454,B 24.9054,C -2.246,E1 25.1472,E2 112.7724} C_DIS
LIN {X 67.8668,Y -30.6717,Z 78,A -29.6549,B 24.9026,C -2.2782,E1 25.1458,E2 114.0982} C_DIS
LIN {X 66.3325,Y -33.8622,Z 78,A -32.4437,B 24.9035,C -2.2681,E1 25.1424,E2 116.8957} C_DIS
LIN {X 65.1925,Y -36.0099,Z 78,A -34.9805,B 24.9056,C -2.2431,E1 25.139,E2 119.4784} C_DIS
LIN {X 63.1521,Y -39.4775,Z 78,A -37.8043,B 24.9056,C -2.2422,E1 25.1349,E2 122.2897} C_DIS
LIN {X 61.5297,Y -41.9621,Z 78,A -40.684,B 24.9077,C -2.2186,E1 25.1303,E2 125.2111} C_DIS
LIN {X 59.2923,Y -45.0695,Z 78,A -44.1008,B 24.9095,C -2.1971,E1 25.1245,E2 128.6623} C_DIS
LIN {X 56.6124,Y -48.3912,Z 78,A -46.4055,B 24.9078,C -2.2168,E1 25.1205,E2 130.9099} C_DIS
LIN {X 54.6494,Y -50.5985,Z 78,A -48.7649,B 24.9085,C -2.2086,E1 25.116,E2 133.2782} C_DIS
LIN {X 52.0651,Y -53.2543,Z 78,A -52.2788,B 24.9106,C -2.1828,E1 25.109,E2 136.8384} C_DIS
LIN {X 49.282,Y -55.8399,Z 78,A -54.4351,B 24.9094,C -2.1979,E1 25.1046,E2 138.9502} C_DIS
LIN {X 46.7392,Y -57.984,Z 78,A -57.1896,B 24.9103,C -2.1868,E1 25.0986,E2 141.7207} C_DIS
LIN {X 43.9773,Y -60.1053,Z 78,A -60.282,B 24.9117,C -2.1695,E1 25.0916,E2 144.8428} C_DIS
LIN {X 41.1249,Y -62.092,Z 78,A -62.1993,B 24.9104,C -2.1856,E1 25.0873,E2 146.7156} C_DIS
LIN {X 39.3487,Y -63.2325,Z 78,A -64.1741,B 24.9115,C -2.1727,E1 25.0825,E2 148.7147} C_DIS
LIN {X 35.4464,Y -65.4997,Z 78,A -67.6395,B 24.9119,C -2.1668,E1 25.0741,E2 152.1839} C_DIS
LIN {X 30.217,Y -68.0717,Z 78,A -71.5458,B 24.9112,C -2.1758,E1 25.0643,E2 156.0585} C_DIS
LIN {X 26.6675,Y -69.5384,Z 78,A -74.7686,B 24.9121,C -2.1642,E1 25.0559,E2 159.3016} C_DIS
LIN {X 23.1666,Y -70.7815,Z 78,A -77.8445,B 24.9129,C -2.1547,E1 25.0477,E2 162.3941} C_DIS
LIN {X 19.9322,Y -71.7601,Z 78,A -80.2256,B 24.9127,C -2.1578,E1 25.0414,E2 164.7637} C_DIS
LIN {X 15.6495,Y -72.8135,Z 78,A -83.4593,B 24.9126,C -2.1589,E1 25.0326,E2 167.9902} C_DIS
LIN {X 11.1891,Y -73.6308,Z 78,A -87.07,B 24.9131,C -2.1529,E1 25.0227,E2 171.6113} C_DIS
LIN {X 8.2746,Y -74.0158,Z 78,A -89.2486,B 24.913,C -2.1537,E1 25.0166,E2 173.7863} C_DIS
LIN {X 4.0287,Y -74.3669,Z 78,A -92.2079,B 24.9124,C -2.1608,E1 25.0084,E2 176.7273} C_DIS
LIN {X 0.4846,Y -74.4612,Z 78,A -93.9311,B 24.9103,C -2.1873,E1 25.0039,E2 178.3872} C_DIS
Enddeposition()
LIN {X 0.4846,Y -74.4612,Z 78,A -93.9311,B 24.9103,C -2.1873,E1 25.0039,E2 178.3872} C_DIS
Startdeposition()
$VEL.CP = VEL_PRINT
LIN {X 3.8892,Y -73.442,Z 78,A -91.346,B 24.909,C -2.2021,E1 25.0111,E2 175.7678} C_DIS
LIN {X 8.4849,Y -73.0537,Z 78,A -88.2127,B 24.9099,C -2.1915,E1 25.0198,E2 172.6615} C_DIS
LIN {X 10.9723,Y -72.7221,Z 78,A -85.0054,B 24.9069,C -2.2272,E1 25.0288,E2 169.3724} C_DIS
LIN {X 15.2656,Y -71.9441,Z 78,A -82.894,B 24.9097,C -2.1945,E1 25.0344,E2 167.3412} C_DIS
LIN {X 19.6725,Y -70.8659,Z 78,A -79.2591,B 24.9091,C -2.2008,E1 25.0443,E2 163.6968} C_DIS
LIN {X 22.4747,Y -70.0267,Z 78,A -76.6399,B 24.9081,C -2.2129,E1 25.0513,E2 161.0537} C_DIS
LIN {X 26.8832,Y -68.4552,Z 78,A -72.8423,B 24.9074,C -2.222,E1 25.0613,E2 157.2426} C_DIS
LIN {X 29.5815,Y -67.3335,Z 78,A -69.9288,B 24.9056,C -2.2435,E1 25.0688,E2 154.2854} C_DIS
LIN {X 33.4423,Y -65.5015,Z 78,A -67.6971,B 24.9077,C -2.2177,E1 25.0742,E2 152.1209} C_DIS
LIN {X 36.944,Y -63.5931,Z 78,A -64.1392,B 24.9062,C -2.2359,E1 25.083,E2 148.5303} C_DIS
LIN {X 40.414,Y -61.4454,Z 78,A -61.1523,B 24.9062,C -2.2365,E1 25.09,E2 145.5517} C_DIS
LIN {X 43.708,Y -59.1484,Z 78,A -58.4147,B 24.9066,C -2.2316,E1 25.0961,E2 142.8352} C_DIS
LIN {X 45.476,Y -57.7995,Z 78,A -56.1549,B 24.905,C -2.2505,E1 25.1012,E2 140.539} C_DIS
LIN {X 48.0047,Y -55.7184,Z 78,A -52.6839,B 24.9022,C -2.2831,E1 25.1087,E2 137.0045} C_DIS
LIN {X 51.7109,Y -52.2955,Z 78,A -50.6512,B 24.9061,C -2.2371,E1 25.1125,E2 135.0891} C_DIS
LIN {X 53.6829,Y -50.2693,Z 78,A -47.6167,B 24.9036,C -2.2666,E1 25.1185,E2 131.9981} C_DIS
LIN {X 55.4706,Y -48.2893,Z 78,A -45.3975,B 24.9028,C -2.276,E1 25.1226,E2 129.7667} C_DIS
LIN {X 58.0767,Y -45.1222,Z 78,A -42.678,B 24.9033,C -2.2704,E1 25.1273,E2 127.0731} C_DIS
LIN {X 59.9987,Y -42.5327,Z 78,A -39.9613,B 24.9022,C -2.2832,E1 25.1317,E2 124.3392} C_DIS
Enddeposition()
END
